// TwinCAT 3 PLC project PLC
// ProgramVersion: 3.1.4024.0
// libraries:
//   EfficientIO Communicator, * (EfficientIO)
//   EfficientIO Energy Basic, * (EfficientIO)
//   Lynus Persistent Data V1, * (Lynus AG)
//   Lynus Standards, * (EfficientIO)
//   Tc2_ModbusSrv, * (Beckhoff Automation GmbH)
//   Tc2_Standard, * (Beckhoff Automation GmbH)
//   Tc2_System, * (Beckhoff Automation GmbH)
//   Tc2_TcpIp, * (Beckhoff Automation GmbH)
//   Tc2_Utilities, * (Beckhoff Automation GmbH)
//   Tc3_Module, * (Beckhoff Automation GmbH)
//   EfficientIO ModbusTCP,1.0.0.9,EfficientIO
// project tree:
//   / FastTask.TcTTO, MiddleTask.TcTTO, SlowTask.TcTTO
//   FB/ fb_Convert4BytesToLreal.TcPOU, FB_IntervalBit.TcPOU (not stored), FB_TCPModbusRequest_PV.TcPOU, FB_TCPModbusRequest_PV_Huawei_inclWrite.TcPOU, FB_TCPModbusRequest_PV_Huawei_inclWrite_oneTurn.TcPOU
//   POUs/ prgBattery.TcPOU, prgComEffIO.TcPOU, prgCS.TcPOU, prgEM.TcPOU, prgEMS.TcPOU, prgGrid.TcPOU, prgPersistent.TcPOU, prgPV_shared.TcPOU, prgPV_separate.TcPOU, prgPV.TcPOU, prgRWEffIO.TcPOU, prgVarEffIO.TcPOU
// real-time tasks:
//   TASK FastTask: cycle T#5ms, priority 19, ADS port 351
//   TASK MiddleTask: cycle T#10ms, priority 20, ADS port 352
//   TASK SlowTask: cycle T#20ms, priority 21, ADS port 353
// I/O:
//   DEVICE Gerät 2 (CX-BK)
//     Box 1 (CX-BK)
// variable links:
//   PLC/PLC Instance <-> Device 2 (CX-BK)/Box 1 (CX-BK)
//     FastTask Inputs/prgGrid.fbKBusState.uiKBusState_OUT <-> Inputs/State
//     MiddleTask Inputs/prgGrid.fbEM1.fbKL3403.byStateCH1 <-> Term 4 (KL3403)/Channel 1/Status
//     MiddleTask Inputs/prgGrid.fbEM1.fbKL3403.byStateCH2 <-> Term 4 (KL3403)/Channel 2/Status
//     MiddleTask Inputs/prgGrid.fbEM1.fbKL3403.byStateCH3 <-> Term 4 (KL3403)/Channel 3/Status
//     MiddleTask Inputs/prgGrid.fbEM1.fbKL3403.iDataInCH1 <-> Term 4 (KL3403)/Channel 1/Daten Ein
//     MiddleTask Inputs/prgGrid.fbEM1.fbKL3403.iDataInCH2 <-> Term 4 (KL3403)/Channel 2/Daten Ein
//     MiddleTask Inputs/prgGrid.fbEM1.fbKL3403.iDataInCH3 <-> Term 4 (KL3403)/Channel 3/Daten Ein
//     MiddleTask Outputs/prgGrid.fbEM1.fbKL3403.byCntrCH1 <-> Term 4 (KL3403)/Channel 1/Kontrolle
//     MiddleTask Outputs/prgGrid.fbEM1.fbKL3403.byCntrCH2 <-> Term 4 (KL3403)/Channel 2/Kontrolle
//     MiddleTask Outputs/prgGrid.fbEM1.fbKL3403.byCntrCH3 <-> Term 4 (KL3403)/Channel 3/Kontrolle

CONFIGURATION PLC
    RESOURCE PLC ON TwinCAT3
        TASK FastTask(INTERVAL := T#5ms, PRIORITY := 19);
        TASK MiddleTask(INTERVAL := T#10ms, PRIORITY := 20);
        TASK SlowTask(INTERVAL := T#20ms, PRIORITY := 21);
        PROGRAM prgPersistent WITH FastTask : prgPersistent;
        PROGRAM prgRWEffIO WITH FastTask : prgRWEffIO;
        PROGRAM prgVarEffIO WITH FastTask : prgVarEffIO;
        PROGRAM prgGrid WITH MiddleTask : prgGrid;
        PROGRAM prgEMS WITH MiddleTask : prgEMS;
        PROGRAM prgCS WITH MiddleTask : prgCS;
        PROGRAM prgEM WITH MiddleTask : prgEM;
        PROGRAM prgBattery WITH MiddleTask : prgBattery;
        PROGRAM prgPV WITH MiddleTask : prgPV;
        PROGRAM prgComEffIO WITH SlowTask : prgComEffIO;
    END_RESOURCE
END_CONFIGURATION

// ---- POUs/prgPersistent.TcPOU
PROGRAM prgPersistent
VAR
	fbUSV		: FB_WritePersistentData_CX81xx;
	
	fb_Reboot		: NT_reboot;
	m_Reboot		: BOOL:=FALSE;
	
	uinit_KbusState: UINT;						//{#lynus.ag#()}
END_VAR

fbUSV(
	eSaveModeData:= eUSVSaveMode.eSaveOnBoth, 
	bLoadPersistentDataOk=> , 
	bPowerFailDetect=> , 
	bError=> , 
	bySaveProcess=> , 
	dwStorageLast24h=> , 
	udiErrorCode=> );
	
	
fb_Reboot(	netid := '',
			delay := 2,
			start := m_Reboot);
	
uinit_KbusState := prgGrid.fbKBusState.uiKBusState_OUT;

END_PROGRAM

// ---- POUs/prgGrid.TcPOU
PROGRAM prgGrid
VAR
	fbKBusState					: FB_K_Bus_State;
	fbEM1						: FB_EM_Beckhoff_KL3403;
	lrPowerGrid					: LREAL;							//{#lynus.ag#()}
	lrPowerEM1_1				: LREAL;							//{#lynus.ag#()}
	lrPowerEM1_2				: LREAL;							//{#lynus.ag#()}
	lrPowerEM1_3				: LREAL;							//{#lynus.ag#()}
	lrCounterGridCon			: LREAL;							//{#lynus.ag#()}
	lrCounterGridProd			: LREAL;							//{#lynus.ag#()}
	lr_GridVoltageL1N_V			: LREAL;							//{#lynus.ag#()}
	lr_GridVoltageL2N_V			: LREAL;							//{#lynus.ag#()}
	lr_GridVoltageL3N_V			: LREAL;							//{#lynus.ag#()}

	lrReactivePowerGrid			: LREAL;							//{#lynus.ag#()}
	lrApparentPowerGrid			: LREAL;							//{#lynus.ag#()}
	fbGrid: FB_Grid_Power;
	lrPowerGrid_cons			: LREAL;							//{#lynus.ag#()}
	lrPowerGrid_prod			: LREAL;							//{#lynus.ag#()}
	lrHouse						: LREAL;							//{#lynus.ag#()}
	
END_VAR

VAR PERSISTENT
	rSizeGridDelivery			: REAL;								//{#lynus.ag#()}
	rSizeGridConn				: REAL;								//{#lynus.ag#()}
END_VAR

//The mapping of this function must be linked with the K-Bus State in the E/A Part
fbKBusState(	uiKBusState_OUT=> , 	
				b_Kbus_notOk=> , 
				word_ErrorCount=> );

//The mapping of this function must be linked with the KL3403 in the E/A Part
//UV1
fbEM1(
	bEnable:= TRUE, 
	bChannel1Invers:= FALSE,				//Invert power data when transformer are mounted upside down
	bChannel2Invers:= FALSE,
	bChannel3Invers:= FALSE,
	uiCurrentTransformerRatioL1:= 1500, // 30 0 / 1 A CTs mounted
	uiCurrentTransformerRatioL2:= 1500, 
	uiCurrentTransformerRatioL3:= 1500, 
	uiKBusState_IN:= fbKBusState.uiKBusState_OUT, 
	stDataEMPower=> , 
	stDataEMCounter=> , 
	stDataEMPowerRealTime=> , 
	stDataEMCounterRealTime=> , 
	diNrOfEM_OUT=> );

lrPowerGrid := fbEM1.stDataEMPower.lrPowerTotal;
lrCounterGridCon := fbEM1.stDataEMCounter.lrTotalCounterEnergy_Consumption;	
lrCounterGridProd := fbEM1.stDataEMCounter.lrTotalCounterEnergy_Production;	
lrPowerEM1_1 := fbEM1.stDataEMPower.lrPowerL1;
lrPowerEM1_2 := fbEM1.stDataEMPower.lrPowerL2;
lrPowerEM1_3 := fbEM1.stDataEMPower.lrPowerL3;

lrReactivePowerGrid:=fbEM1.stDataEMPower.lrReactivePowerTotal;
lrApparentPowerGrid:=fbEM1.stDataEMPower.lrApparentPowerTotal;

lr_GridVoltageL1N_V:=fbEM1.stDataEMPower.lrVoltageL1N;
lr_GridVoltageL2N_V:=fbEM1.stDataEMPower.lrVoltageL2N;
lr_GridVoltageL3N_V:=fbEM1.stDataEMPower.lrVoltageL3N;

fbGrid(
	bEnable:= TRUE, 
	diNrOfEMS_IN:= prgEMS.fbEMS.diNrOfEMS_OUT, 
	diNrOfEM_IN_Grid:= 	fbEM1.diNrOfEM_OUT,			//prgBattery.fbBattery.diNrOfEM_OUT_Grid, 
	rSizeGridConn:= rSizeGridConn, 
	stDataGrid=> , 
	diNrOfGrid_OUT=> );

lrPowerGrid_cons 	:= 	fbEM1.stDataEMPower.lrPowerConsumption;
lrPowerGrid_prod	:= 	fbEM1.stDataEMPower.lrPowerProduction;

lrHouse := lrPowerGrid + prgPV.lrPowerPV - prgCS.lrPowerCS + prgBattery.lrPowerBattery + prgEM.lrPower_Fuse - prgEM.lrPower_Fuse_EM2 - prgEM.lrPower_Fuse_EM3;

END_PROGRAM

// ---- POUs/prgEMS.TcPOU
PROGRAM prgEMS
VAR PERSISTENT
	byMaxDepthOfDischrgEPO		: BYTE;							//{#lynus.ag#()}
	byPrioMinChrgBattSOCInEPO	: BYTE;							//{#lynus.ag#()}
	byResChrgfromGridToBatt		: BYTE;							//{#lynus.ag#()}
	byReserveSOCEPO				: BYTE;							//{#lynus.ag#()}
	uiUpdateTime				: UINT;							//{#lynus.ag#()}
	bEnableEMS					: BOOL;							//{#lynus.ag#()}
	bAllowChrgFromGrid			: BOOL;							//{#lynus.ag#()}
	bActivateMainFuse			: BOOL;							//{#lynus.ag#()}
	rMainFuseCSEMS				: REAL;							//{#lynus.ag#()}
	iOperationModeEMS			: INT;							//{#lynus.ag#()}
	by_MinSOC_AdaptiveLC		: BYTE;							//{#lynus.ag#()}
END_VAR
VAR
	fbEMS						: FB_EMS_V12;
	bIsEnableEMS				: BOOL;							//{#lynus.ag#()}
	bStateAllowChrgFromGrid		: BOOL;							//{#lynus.ag#()}
	bHPActivate					: BOOL;							//{#lynus.ag#()}
	bControllingState			: BOOL;							//{#lynus.ag#()}
	bSActivateMainFuse			: BOOL;							//{#lynus.ag#()}
	iMessageEMS					: INT;							//{#lynus.ag#()}
	rHeartbeatEMS				: REAL;							//{#lynus.ag#()}
	rErrorWarningEMS			: REAL;							//{#lynus.ag#()}
	rReadyEMS					: REAL;							//{#lynus.ag#()}
	rNewBatteryPowerEMS			: REAL;							//{#lynus.ag#()}
	b_Chargefor3Hours			: BOOL;							//{#lynus.ag#()}
	b_Chargefor3Hours_Active	: BOOL;							//{#lynus.ag#()}
	b_Chargefor1Hour			: BOOL;							//{#lynus.ag#()}
	b_Chargefor1Hour_Active		: BOOL;							//{#lynus.ag#()}
	ton_ChargeTimer_3hours		: ton;
	ton_ChargeTimer_1hour		: ton;
	rs_charge_3hours			: rs;
	rs_charge_1hour				: rs;
	r_trig_Charge_3hours		: R_trig;
	r_trig_Charge_1hour			: R_trig;
	fb_Meter	:	FB_EM_Electric_3P_Ext_Input;
	iOperationModeEMS_actual			: INT;							//{#lynus.ag#()}
	di_temp : DINT;
	m_ZeroPowerRegulationActive: BOOL:=FALSE;						//{#lynus.ag#()}
	timer_CarConnected_CSPowerlow: Ton;

END_VAR

fbEMS.stSetupEMS.bAllowChrgFromGrid := bAllowChrgFromGrid;
fbEMS.stSetupEMS.byMaxDepthOfDischrgEPO := byMaxDepthOfDischrgEPO;
fbEMS.stSetupEMS.byResChrgfromGridToBatt := byResChrgfromGridToBatt;
fbEMS.stSetupEMS.byPrioMinChrgBattSOCInEPO := byPrioMinChrgBattSOCInEPO;
fbEMS.stSetupEMS.byReserveSOCEPO := SEL(b_Chargefor3Hours_Active OR b_Chargefor1Hour_Active,byReserveSOCEPO,100);
fbEMS.stSetupEMS.rSizeMainFuseCS := rMainFuseCSEMS;
fbEMS.stSetupEMS.uiUpdateTime := uiUpdateTime;
fbEMS.stSetupEMS.bEnableMainFuseFunction := bActivateMainFuse;

IF iOperationModeEMS = 0 THEN 
	fbEMS.eOperationMode_Ext := E_OperatingMode_EMS.eAllOff;
ELSIF iOperationModeEMS = 1 THEN 
	fbEMS.eOperationMode_Ext := E_OperatingMode_EMS.eSelfConsumption;	
ELSIF iOperationModeEMS = 2 THEN 
	fbEMS.eOperationMode_Ext := E_OperatingMode_EMS.ePeakLoadCapping;
ELSIF iOperationModeEMS = 3 THEN 
	fbEMS.eOperationMode_Ext := E_OperatingMode_EMS.eLoadManagement;			
ELSIF iOperationModeEMS = 4 THEN 
	fbEMS.eOperationMode_Ext := E_OperatingMode_EMS.eAdaptiveLoadControl;		
END_IF
di_temp := fbEMS.diNumberOfActiveBatterys;

fbEMS(
	diNrOfEM_IN_ECS:= , 
	stSetupEMS:= , 
	eOperationMode_Ext:= , 
	eSpeedModeBackendController:= E_SpeedModeBackendController_EMS.eSlow,	//.efast, 
	eSpeedModeLocalController:= E_SpeedModeLocalController_EMS.eSlow,    //efast,
	bZeroPowerRegulation	:= m_ZeroPowerRegulationActive, 
	by_MinSOC_AdaptiveLC:= by_MinSOC_AdaptiveLC, 
	bActivateHP:= bHPActivate, 
	bControllingState:= TRUE, //bControllingState, 
	rHeartbeat:= rHeartbeatEMS, 
	rErrorWarning:= rErrorWarningEMS, 
	rEnergyOptReady:= rReadyEMS, 
	rNewBattPower:= rNewBatteryPowerEMS,
	b_AnyCarConnected:= prgCS.bCarConnected and not timer_CarConnected_CSPowerlow.Q ,  
	eMessageEMS=> iMessageEMS, 
	bStateEnable=> bIsEnableEMS, 
	bStateAllowChrgFromGrid=> bStateAllowChrgFromGrid, 
	bMissingPowerData=> , 
	bSurplusAvailable=> , 
	byProgress=> , 
	uiState_OUT=> , 
	diNrOfEMS_OUT=> , 
	arrMinPrioReached=> , 
	arrMaxPrioReached=> );
	
bSActivateMainFuse := fbEMS.stSetupEMS.bEnableMainFuseFunction;	
iOperationModeEMS_actual := fbEMS.eOperationMode;

// charge for 3 hours
r_trig_Charge_3hours (clk := b_Chargefor3Hours);
r_trig_Charge_1hour (clk := b_Chargefor1Hour);


rs_charge_3hours	(	Set := r_trig_Charge_3hours.Q ,
						Reset1 := ton_ChargeTimer_3hours.Q OR (rs_Charge_3hours.Q1 AND r_trig_Charge_3hours.Q),
						Q1 => b_Chargefor3Hours_Active);
rs_charge_1hour		(	Set := r_trig_Charge_1hour.Q ,
						Reset1 := ton_ChargeTimer_1hour.Q OR (rs_Charge_1hour.Q1 AND r_trig_Charge_1hour.Q),
						Q1 => b_Chargefor1Hour_Active);			
ton_ChargeTimer_3hours	( 	IN := rs_charge_3hours.Q1,
							PT := T#3H,
							Q => );
ton_ChargeTimer_1hour	( 	IN := rs_charge_1hour.Q1,
							PT := T#1H,
							Q => );
	

timer_CarConnected_CSPowerlow( 	IN := prgCS.bCarConnected AND prgCS.lrPowerCS < 2,	// required to get out of zero power regulation if a car is connected all night long
								PT := T#10M);
							
m_ZeroPowerRegulationActive := prgCS.bCarConnected AND NOT timer_CarConnected_CSPowerlow.Q;
	

fb_Meter(
	bEnable:= TRUE, 
	bPowerDataInvers:= , 
	bErrorExt:= , 
	bWarningExt:= , 
	lrTotalCounterEnergy_Consumption:= , 
	lrTotalCounterEnergy_Production:= , 
	lrCounterEnergyT1_Consumption:= , 
	lrCounterEnergyT2_Consumption:= , 
	lrCounterEnergyT1_Production:= , 
	lrCounterEnergyT2_Production:= , 
	lrCurrentL1:= , 
	lrVoltageL1N:= , 
	lrVoltageL1L2:= , 
	lrPowerL1:= , 
	lrCurrentL2:= , 
	lrVoltageL2N:= , 
	lrVoltageL2L3:= , 
	lrPowerL2:= , 
	lrCurrentL3:= , 
	lrVoltageL3N:= , 
	lrVoltageL3L1:= , 
	lrPowerL3:= , 
	lrPowerTotal:= prgEM.lrPower_Fuse,
	lrFrequency:= , 
	lrReactivePowerTotal:= , 
	lrApparentPowerTotal:= , 
	stDataEMPower=> , 
	stDataEMCounter=> , 
	diNrOfEM_OUT=> );		// da gehört was hin, damit er auf die fuseline regeln kann

END_PROGRAM

// ---- POUs/prgCS.TcPOU
PROGRAM prgCS
VAR PERSISTENT
	bEnabledCS				: BOOL;									//{#lynus.ag#()}
	byPrioCS				: BYTE;									//{#lynus.ag#()}
	bySOC_E_CS				: BYTE;									//{#lynus.ag#()}
	bySOC_D_CS				: BYTE;									//{#lynus.ag#()}
	byMinPowerCS			: BYTE;									//{#lynus.ag#()}
	rMaxPowerCS				: REAL;									//{#lynus.ag#()}
	lrCounterCS				: LREAL;								//{#lynus.ag#()}
	bManualyOn				: BOOL;									//{#lynus.ag#()}
	byMinPower				: BYTE;									//{#lynus.ag#()}
	byManualyTargetPower	: BYTE;									//{#lynus.ag#()}
	m_ChargingLimit			: BOOL;									//{#lynus.ag#()}
	bOnEmergPowerOff		: BOOL;									//{#lynus.ag#()}
END_VAR
VAR
	fbCS					: FB_ECS_Alpitronic_Hypercharger;
	fbCSCounter				: FB_EnergyCounter;
	bIsEnabledCS			: BOOL;									//{#lynus.ag#()}
	byErrorWarningCS		: BYTE;									//{#lynus.ag#()}
	byStateMinPowerCS		: BYTE;									//{#lynus.ag#()}
	rTargetPowerCS			: REAL;									//{#lynus.ag#()}
	bCarConnected			: BOOL;									//{#lynus.ag#()}
	rChrgTime				: REAL;									//{#lynus.ag#()}
	lrPowerCS				: LREAL;								//{#lynus.ag#()}
	bSManualyOn				: BOOL;									//{#lynus.ag#()}
	bySManualyTargetPower	: BYTE;									//{#lynus.ag#()}
	str_IP: STRING(15):='172.16.127.151';
	rSOC_1					: REAL;									//{#lynus.ag#()}
	rSOC_2					: REAL;									//{#lynus.ag#()}
	bSOnEmergPowerOff		: BOOL;									//{#lynus.ag#()}
END_VAR

fbCS.stSetupECS.byDisableSOC := bySOC_D_CS;
fbCS.stSetupECS.byEnableSOC := bySOC_E_CS;
fbCS.stSetupECS.byPriority := byPrioCS;
fbCS.stSetupECS.rMaxPower := rMaxPowerCS;
fbCS.stSetupECS.byCSMinPower := byMinPowerCS;
fbCS.stSetupECS.bManualyOn := bManualyOn;
fbCS.stSetupECS.byManualyTargetPower := byManualyTargetPower;
fbCS.stSetupECS.byCSMinPower := byMinPower;
fbCS.stSetupECS.bOnEmergPowerOff := bOnEmergPowerOff;

fbCS(
	bEnable:= bEnabledCS, 
	bPowerDataInvers:= ,  
	byUnitID:= 1,				//Allways 1 
	diNrOfEMS_IN:= prgEMS.fbEMS.diNrOfEMS_OUT, 
	diNrOfEM_IN_CS:= , 
	sIPAdress:= str_IP, 
	stSetupECS:= , 
	stDataECS=> , 
	diNrOfECS_OUT=> );

bIsEnabledCS := fbCS.stDataECS.bEnabled;
byStateMinPowerCS := fbCS.stDataECS.bySCSMinPower;
rTargetPowerCS := fbCS.stDataECS.rTargetPower;	
byErrorWarningCS := fbCS.stDataECS.byErrorWarning;
bCarConnected := fbCS.stDataECS.bCarConnected;
rChrgTime := MAX(fbCS.stDataECS.arrChargingTimeInMin[1],fbCS.stDataECS.arrChargingTimeInMin[2]);
lrPowerCS := fbCS.stDataECS.lrTotalPower;
bSManualyOn := fbCS.stDataECS.bSManualyOn;
bSOnEmergPowerOff := fbCS.stDataECS.bSOnEmergPowerOff;

bySManualyTargetPower := fbCS.stDataECS.bySManualyTargetPower;
rSOC_1	:= DWORD_TO_REAL(fbCS.stDataECS.arrSocketSOCCar[1]);
rSOC_2	:= DWORD_TO_REAL(fbCS.stDataECS.arrSocketSOCCar[2]);						

// EnergyCounter
fbCSCounter(
	byActiveTariff:= 1, 
	lrPowerInput:= lrPowerCS, 
	lrTotalCounterEnergy_Consumption=> );
	
IF fbCSCounter.lrTotalCounterEnergy_Consumption > lrCounterCS THEN  	
	lrCounterCS := fbCSCounter.lrTotalCounterEnergy_Consumption;
END_IF

END_PROGRAM

// ---- POUs/prgEM.TcPOU
PROGRAM prgEM
VAR
	// Meter1 - Halle Verteiler
	fb_External_Meter			: fb_EM24_DIN;
	str_IP: STRING(15)			:= '172.16.127.51'	;
	
	lrPower_Fuse				: LREAL;							//{#lynus.ag#()}
	lrPower_Fuse_1				: LREAL;							//{#lynus.ag#()}
	lrPower_Fuse_2				: LREAL;							//{#lynus.ag#()}
	lrPower_Fuse_3				: LREAL;							//{#lynus.ag#()}
	lrCurrent_Fuse_1			: LREAL;							//{#lynus.ag#()}
	lrCurrent_Fuse_2			: LREAL;							//{#lynus.ag#()}
	lrCurrent_Fuse_3			: LREAL;							//{#lynus.ag#()}
	lrCounter_Fuse_Con			: LREAL;							//{#lynus.ag#()}
	lrCounter_Fuse_Prod			: LREAL;							//{#lynus.ag#()}
	lr_Voltage_Fuse_L1N_V		: LREAL;							//{#lynus.ag#()}
	lr_Voltage_Fuse_L2N_V		: LREAL;							//{#lynus.ag#()}
	lr_Voltage_Fuse_L3N_V		: LREAL;							//{#lynus.ag#()}
	lr_Voltage_Fuse_L1L2_V		: LREAL;							//{#lynus.ag#()}
	lr_Voltage_Fuse_L2L3_V		: LREAL;							//{#lynus.ag#()}
	lr_Voltage_Fuse_L3L1_V		: LREAL;							//{#lynus.ag#()}

	lrReactivePowerFuse			: LREAL;							//{#lynus.ag#()}
	lrApparentPowerFuse			: LREAL;							//{#lynus.ag#()}
	m_invert					: BOOL:=TRUE;
	
	
	// Meter2 - 3. Stock
	fb_External_Meter_2				: fb_EM24_DIN;
	str_IP_EM2						: STRING(15):= '172.16.127.52'	;
	
	lrPower_Fuse_EM2				: LREAL;							//{#lynus.ag#()}
	lrPower_Fuse_1_EM2				: LREAL;							//{#lynus.ag#()}
	lrPower_Fuse_2_EM2				: LREAL;							//{#lynus.ag#()}
	lrPower_Fuse_3_EM2				: LREAL;							//{#lynus.ag#()}
	lrCurrent_Fuse_1_EM2			: LREAL;							//{#lynus.ag#()}
	lrCurrent_Fuse_2_EM2			: LREAL;							//{#lynus.ag#()}
	lrCurrent_Fuse_3_EM2			: LREAL;							//{#lynus.ag#()}
	lrCounter_Fuse_Con_EM2			: LREAL;							//{#lynus.ag#()}
	lrCounter_Fuse_Prod_EM2			: LREAL;							//{#lynus.ag#()}
	lr_Voltage_Fuse_L1N_V_EM2		: LREAL;							//{#lynus.ag#()}
	lr_Voltage_Fuse_L2N_V_EM2		: LREAL;							//{#lynus.ag#()}
	lr_Voltage_Fuse_L3N_V_EM2		: LREAL;							//{#lynus.ag#()}
	lr_Voltage_Fuse_L1L2_V_EM2		: LREAL;							//{#lynus.ag#()}
	lr_Voltage_Fuse_L2L3_V_EM2		: LREAL;							//{#lynus.ag#()}
	lr_Voltage_Fuse_L3L1_V_EM2		: LREAL;							//{#lynus.ag#()}

	lrReactivePowerFuse_EM2			: LREAL;							//{#lynus.ag#()}
	lrApparentPowerFuse_EM2			: LREAL;							//{#lynus.ag#()}
	m_invert_EM2					: BOOL:=FALSE;
	
	
	// Meter3 - EG
	fb_External_Meter_3				: fb_EM24_DIN;
	str_IP_EM3						: STRING(15):= '172.16.127.53'	;
	
	lrPower_Fuse_EM3				: LREAL;							//{#lynus.ag#()}
	lrPower_Fuse_1_EM3				: LREAL;							//{#lynus.ag#()}
	lrPower_Fuse_2_EM3				: LREAL;							//{#lynus.ag#()}
	lrPower_Fuse_3_EM3				: LREAL;							//{#lynus.ag#()}
	lrCurrent_Fuse_1_EM3			: LREAL;							//{#lynus.ag#()}
	lrCurrent_Fuse_2_EM3			: LREAL;							//{#lynus.ag#()}
	lrCurrent_Fuse_3_EM3			: LREAL;							//{#lynus.ag#()}
	lrCounter_Fuse_Con_EM3			: LREAL;							//{#lynus.ag#()}
	lrCounter_Fuse_Prod_EM3			: LREAL;							//{#lynus.ag#()}
	lr_Voltage_Fuse_L1N_V_EM3		: LREAL;							//{#lynus.ag#()}
	lr_Voltage_Fuse_L2N_V_EM3		: LREAL;							//{#lynus.ag#()}
	lr_Voltage_Fuse_L3N_V_EM3		: LREAL;							//{#lynus.ag#()}
	lr_Voltage_Fuse_L1L2_V_EM3		: LREAL;							//{#lynus.ag#()}
	lr_Voltage_Fuse_L2L3_V_EM3		: LREAL;							//{#lynus.ag#()}
	lr_Voltage_Fuse_L3L1_V_EM3		: LREAL;							//{#lynus.ag#()}

	lrReactivePowerFuse_EM3			: LREAL;							//{#lynus.ag#()}
	lrApparentPowerFuse_EM3			: LREAL;							//{#lynus.ag#()}
	m_invert_EM3					: BOOL:=FALSE;
	
END_VAR

// Meter1 - Halle Verteiler
fb_External_Meter(
	m_Enable:= TRUE, 
	str_IPAdress:= str_IP, 
	real_RealPower_kW=> lrPower_Fuse, 
	real_RealPowerL1_kW=> lrPower_Fuse_1, 
	real_RealPowerL2_kW=> lrPower_Fuse_2, 
	real_RealPowerL3_kW=> lrPower_Fuse_3, 
	real_ReactivePower_kVAr=> lrReactivePowerFuse, 
	real_ApparentPower_kVA=> lrApparentPowerFuse, 
	real_Frequency_Hz=> , 
	real_VoltageL1N_V=> lr_Voltage_Fuse_L1N_V, 
	real_VoltageL2N_V=> lr_Voltage_Fuse_L2N_V, 
	real_VoltageL3N_V=> lr_Voltage_Fuse_L3N_V, 
	real_VoltageL1L2_V=> lr_Voltage_Fuse_L1L2_V, 
	real_VoltageL2L3_V=> lr_Voltage_Fuse_L2L3_V, 
	real_VoltageL3L1_V=> lr_Voltage_Fuse_L3L1_V, 
	real_CurrentL1_A=> lrCurrent_Fuse_1, 
	real_CurrentL2_A=> lrCurrent_Fuse_2, 
	real_CurrentL3_A=> lrCurrent_Fuse_3, 
	real_EnergyTotal_Import_kWh=> , 
	real_EnergyTotal_Export_kWh=> , 
	real_EnergyTotal_ExportT1_kWh=> , 
	real_EnergyTotal_ExportT2_kWh=> , 
	real_EnergyTotal_ExportT3_kWh=> , 
	real_EnergyTotal_ExportT4_kWh=> , 
	m_PollSuccessful=> , 
	udint_Error_ID=> );
IF m_invert THEN
	lrPower_Fuse_1 		:= -lrPower_Fuse_1 		;
    lrPower_Fuse_2      := -lrPower_Fuse_2      ;
    lrPower_Fuse_3      := -lrPower_Fuse_3      ;
	lrPower_Fuse        := -lrPower_Fuse        ;
	lrCurrent_Fuse_1    := -lrCurrent_Fuse_1    ;
    lrCurrent_Fuse_2    := -lrCurrent_Fuse_2    ;
    lrCurrent_Fuse_3    := -lrCurrent_Fuse_3    ;
END_IF	
IF lrPower_Fuse > 0 THEN 
	lrCounter_Fuse_Con := lrPower_Fuse;
	lrCounter_Fuse_Prod := 0;
ELSE
	lrCounter_Fuse_Prod := lrPower_Fuse;
	lrCounter_Fuse_Con := 0;
END_IF


// Meter2 - 3. Stock
fb_External_Meter_2(
	m_Enable:= TRUE, 
	str_IPAdress:= str_IP_EM2, 
	real_RealPower_kW=> lrPower_Fuse_EM2, 
	real_RealPowerL1_kW=> lrPower_Fuse_1_EM2, 
	real_RealPowerL2_kW=> lrPower_Fuse_2_EM2, 
	real_RealPowerL3_kW=> lrPower_Fuse_3_EM2, 
	real_ReactivePower_kVAr=> lrReactivePowerFuse_EM2, 
	real_ApparentPower_kVA=> lrApparentPowerFuse_EM2, 
	real_Frequency_Hz=> , 
	real_VoltageL1N_V=> lr_Voltage_Fuse_L1N_V_EM2, 
	real_VoltageL2N_V=> lr_Voltage_Fuse_L2N_V_EM2, 
	real_VoltageL3N_V=> lr_Voltage_Fuse_L3N_V_EM2, 
	real_VoltageL1L2_V=> lr_Voltage_Fuse_L1L2_V_EM2, 
	real_VoltageL2L3_V=> lr_Voltage_Fuse_L2L3_V_EM2, 
	real_VoltageL3L1_V=> lr_Voltage_Fuse_L3L1_V_EM2, 
	real_CurrentL1_A=> lrCurrent_Fuse_1_EM2, 
	real_CurrentL2_A=> lrCurrent_Fuse_2_EM2, 
	real_CurrentL3_A=> lrCurrent_Fuse_3_EM2, 
	real_EnergyTotal_Import_kWh=> , 
	real_EnergyTotal_Export_kWh=> , 
	real_EnergyTotal_ExportT1_kWh=> , 
	real_EnergyTotal_ExportT2_kWh=> , 
	real_EnergyTotal_ExportT3_kWh=> , 
	real_EnergyTotal_ExportT4_kWh=> , 
	m_PollSuccessful=> , 
	udint_Error_ID=> );
IF m_invert_EM2 THEN
	lrPower_Fuse_1_EM2 		:= -lrPower_Fuse_1_EM2 		;
    lrPower_Fuse_2_EM2      := -lrPower_Fuse_2_EM2      ;
    lrPower_Fuse_3_EM2      := -lrPower_Fuse_3_EM2      ;
	lrPower_Fuse_EM2        := -lrPower_Fuse_EM2        ;
	lrCurrent_Fuse_1_EM2    := -lrCurrent_Fuse_1_EM2    ;
    lrCurrent_Fuse_2_EM2    := -lrCurrent_Fuse_2_EM2    ;
    lrCurrent_Fuse_3_EM2    := -lrCurrent_Fuse_3_EM2    ;
END_IF	
IF lrPower_Fuse_EM2 > 0 THEN 
	lrCounter_Fuse_Con_EM2 := lrPower_Fuse_EM2;
	lrCounter_Fuse_Prod_EM2 := 0;
ELSE
	lrCounter_Fuse_Prod_EM2 := lrPower_Fuse_EM2;
	lrCounter_Fuse_Con_EM2 := 0;
END_IF


// Meter3 - EG
fb_External_Meter_3(
	m_Enable:= TRUE, 
	str_IPAdress:= str_IP_EM3, 
	real_RealPower_kW=> lrPower_Fuse_EM3, 
	real_RealPowerL1_kW=> lrPower_Fuse_1_EM3, 
	real_RealPowerL2_kW=> lrPower_Fuse_2_EM3, 
	real_RealPowerL3_kW=> lrPower_Fuse_3_EM3, 
	real_ReactivePower_kVAr=> lrReactivePowerFuse_EM3, 
	real_ApparentPower_kVA=> lrApparentPowerFuse_EM3, 
	real_Frequency_Hz=> , 
	real_VoltageL1N_V=> lr_Voltage_Fuse_L1N_V_EM3, 
	real_VoltageL2N_V=> lr_Voltage_Fuse_L2N_V_EM3, 
	real_VoltageL3N_V=> lr_Voltage_Fuse_L3N_V_EM3, 
	real_VoltageL1L2_V=> lr_Voltage_Fuse_L1L2_V_EM3, 
	real_VoltageL2L3_V=> lr_Voltage_Fuse_L2L3_V_EM3, 
	real_VoltageL3L1_V=> lr_Voltage_Fuse_L3L1_V_EM3, 
	real_CurrentL1_A=> lrCurrent_Fuse_1_EM3, 
	real_CurrentL2_A=> lrCurrent_Fuse_2_EM3, 
	real_CurrentL3_A=> lrCurrent_Fuse_3_EM3, 
	real_EnergyTotal_Import_kWh=> , 
	real_EnergyTotal_Export_kWh=> , 
	real_EnergyTotal_ExportT1_kWh=> , 
	real_EnergyTotal_ExportT2_kWh=> , 
	real_EnergyTotal_ExportT3_kWh=> , 
	real_EnergyTotal_ExportT4_kWh=> , 
	m_PollSuccessful=> , 
	udint_Error_ID=> );
IF m_invert_EM3 THEN
	lrPower_Fuse_1_EM3 		:= -lrPower_Fuse_1_EM3 		;
    lrPower_Fuse_2_EM3      := -lrPower_Fuse_2_EM3      ;
    lrPower_Fuse_3_EM3      := -lrPower_Fuse_3_EM3      ;
	lrPower_Fuse_EM3        := -lrPower_Fuse_EM3        ;
	lrCurrent_Fuse_1_EM3    := -lrCurrent_Fuse_1_EM3    ;
    lrCurrent_Fuse_2_EM3    := -lrCurrent_Fuse_2_EM3    ;
    lrCurrent_Fuse_3_EM3    := -lrCurrent_Fuse_3_EM3    ;
END_IF	
IF lrPower_Fuse_EM3 > 0 THEN 
	lrCounter_Fuse_Con_EM3 := lrPower_Fuse_EM3;
	lrCounter_Fuse_Prod_EM3 := 0;
ELSE
	lrCounter_Fuse_Prod_EM3 := lrPower_Fuse_EM3;
	lrCounter_Fuse_Con_EM3 := 0;
END_IF

END_PROGRAM

// ---- POUs/prgPV.TcPOU
PROGRAM prgPV
VAR
	lrPowerPV				: LREAL;				//{#lynus.ag#()}
		// extend or reduce amount of PV Inverters
	lrPowerPV_1				: LREAL;				//{#lynus.ag#()}
	lrPowerPV_2				: LREAL;				//{#lynus.ag#()}
	uint_setPoint_onetenth: UINT;						//{#lynus.ag#()}

	m_shared: BOOL;
END_VAR
VAR PERSISTENT
	lrCounterPV_1				: LREAL;				//{#lynus.ag#()}
	lrCounterPV_2				: LREAL;				//{#lynus.ag#()}
END_VAR

IF m_shared THEN
	prgPV_shared();
	lrPowerPV 				:= prgPV_shared.lrPowerPV;
	lrPowerPV_1 			:= prgPV_shared.lrPowerPV_1;
	lrPowerPV_2 			:= prgPV_shared.lrPowerPV_2;
	uint_setPoint_onetenth 	:= prgPV_shared.uint_setPoint_onetenth;
	lrCounterPV_1			:= prgPV_shared.lrCounterPV_1;
	lrCounterPV_2			:= prgPV_shared.lrCounterPV_2;
ELSE
	prgPV_separate();
	lrPowerPV 				:= prgPV_separate.lrPowerPV;
	lrPowerPV_1 			:= prgPV_separate.lrPowerPV_1;
	lrPowerPV_2 			:= prgPV_separate.lrPowerPV_2;
	uint_setPoint_onetenth 	:= prgPV_separate.uint_setPoint_onetenth;
	lrCounterPV_1			:= prgPV_separate.lrCounterPV_1;
	lrCounterPV_2			:= prgPV_separate.lrCounterPV_2;
END_IF

END_PROGRAM

// ---- POUs/prgPV_shared.TcPOU
PROGRAM prgPV_shared
VAR
	fbPVCounter_1			: FB_EnergyCounter;
	fbPVCounter_2			: FB_EnergyCounter;
	lrPowerPV				: LREAL;				
		// extend or reduce amount of PV Inverters
	lrPowerPV_1				: LREAL;				
	lrPowerPV_2				: LREAL;				

	str_IP: STRING(15) := '172.16.127.240';
	FB_PV_1:FB_TCPModbusRequest_PV_Huawei_inclWrite;	
	FB_PV_2:FB_TCPModbusRequest_PV_Huawei_inclWrite;	
	fb_Meter_1		: FB_EM_Electric_3P_Ext_Input;
	fbPVInt_1		: FB_PV_Power;
	fb_Meter_2		: FB_EM_Electric_3P_Ext_Input;
	fbPVInt_2		: FB_PV_Power;
	

	FB_PID_Inverter :FB_PID;

	uint_setPoint_onetenth: UINT;					

	rPValue: REAL := 0.5;
	udint_IValue: UDINT:=250;
	udint_DValue: UDINT:=30;

	unit_Temp: UINT;
	real_max: REAL:=1000;
	real_min: REAL:=10;

END_VAR
VAR PERSISTENT
	lrCounterPV_1				: LREAL;				
	lrCounterPV_2				: LREAL;				
	m_Direction: BOOL := true;
END_VAR

FB_PV_1(
	b_Enable:= , 
	by_slave_ID:= 1, 
	str_IPAdress:= str_ip, 
	uint_SetPoint_onetenth:= uint_setPoint_onetenth, 
	lreal_RealPower_kW=> lrPowerPV_1,  );


fbPVCounter_1(	byActiveTariff := 1,	
	
				lrPowerInput := 0-lrPowerPV_1,
				lrTotalCounterEnergy_Production => lrCounterPV_1);


FB_PV_2(
	b_Enable:= , 
	by_slave_ID:= 2, 
	str_IPAdress:= str_ip, 
	uint_SetPoint_onetenth:= uint_setPoint_onetenth, 
	lreal_RealPower_kW=> lrPowerPV_2,  );


fbPVCounter_2(	byActiveTariff := 1,	
				lrPowerInput := 0-lrPowerPV_2,
				lrTotalCounterEnergy_Production => lrCounterPV_2);

lrPowerPV := lrPowerPV_1 + lrPowerPV_2;

fbPVInt_1(
	bEnable:= TRUE, 
	bPowerDataInvers:= , 
	diNrOfEM_IN_PV:= fb_Meter_1.diNrOfEM_OUT, 
	stDataPv=> , 
	diNrOfPv_OUT=> );
	
fb_Meter_1(
	bEnable:= TRUE, 
	bPowerDataInvers:= , 
	bErrorExt:= , 
	bWarningExt:= , 
	lrTotalCounterEnergy_Consumption:= , 
	lrTotalCounterEnergy_Production:= , 
	lrCounterEnergyT1_Consumption:= , 
	lrCounterEnergyT2_Consumption:= , 
	lrCounterEnergyT1_Production:= , 
	lrCounterEnergyT2_Production:= , 
	lrCurrentL1:= , 
	lrVoltageL1N:= , 
	lrVoltageL1L2:= , 
	lrPowerL1:= , 
	lrCurrentL2:= , 
	lrVoltageL2N:= , 
	lrVoltageL2L3:= , 
	lrPowerL2:= , 
	lrCurrentL3:= , 
	lrVoltageL3N:= , 
	lrVoltageL3L1:= , 
	lrPowerL3:= , 
	lrPowerTotal:= lrPowerPV_1,
	lrFrequency:= , 
	lrReactivePowerTotal:= , 
	lrApparentPowerTotal:= , 
	stDataEMPower=> , 
	stDataEMCounter=> , 
	diNrOfEM_OUT=> );

	

fbPVInt_2(
	bEnable:= TRUE, 
	bPowerDataInvers:= , 
	diNrOfEM_IN_PV:= fb_Meter_2.diNrOfEM_OUT, 
	stDataPv=> , 
	diNrOfPv_OUT=> );
	
fb_Meter_2(	
	bEnable:= TRUE, 
	bPowerDataInvers:= , 
	bErrorExt:= , 
	bWarningExt:= , 
	lrTotalCounterEnergy_Consumption:= , 
	lrTotalCounterEnergy_Production:= , 
	lrCounterEnergyT1_Consumption:= , 
	lrCounterEnergyT2_Consumption:= , 
	lrCounterEnergyT1_Production:= , 
	lrCounterEnergyT2_Production:= , 
	lrCurrentL1:= , 
	lrVoltageL1N:= , 
	lrVoltageL1L2:= , 
	lrPowerL1:= , 
	lrCurrentL2:= , 
	lrVoltageL2N:= , 
	lrVoltageL2L3:= , 
	lrPowerL2:= , 
	lrCurrentL3:= , 
	lrVoltageL3N:= , 
	lrVoltageL3L1:= , 
	lrPowerL3:= , 
	lrPowerTotal:= lrPowerPV_2,
	lrFrequency:= , 
	lrReactivePowerTotal:= , 
	lrApparentPowerTotal:= , 
	stDataEMPower=> , 
	stDataEMCounter=> , 
	diNrOfEM_OUT=> );

	
FB_PID_Inverter(
		bEnable:= TRUE, 
		rSetpoint:= -prgGrid.rSizeGridDelivery, 
		udiIValue:= udint_IValue, 
		udiDValue:= udint_DValue, 
		udiDamping:= 0, 
		rPValue:= rPValue, 
		rMaxValue:= real_max, 
		rMinValue:= real_min, 
		rNeutralZone:= 1, 
		bDirection:= m_Direction, 
		rActualValue:=  LREAL_TO_REAL(prgGrid.fbEM1.stDataEMPowerRealTime.lrPowerTotal),
		rQController=> );
uint_setPoint_onetenth := REAL_TO_UINT(FB_PID_Inverter.rQController);

END_PROGRAM

// ---- FB/FB_TCPModbusRequest_PV_Huawei_inclWrite.TcPOU
FUNCTION_BLOCK FB_TCPModbusRequest_PV_Huawei_inclWrite
VAR_INPUT
	b_Enable: BOOL;
	by_slave_ID	:BYTE;
	str_IPAdress: STRING(15);
	uint_SetPoint_onetenth	:UINT;
END_VAR
VAR_OUTPUT

	lreal_RealPower_kW:LREAL;
	lreal_Voltage_L1L2_V: LREAL;
	lreal_Voltage_L2L3_V: LREAL;
	lreal_Voltage_L3L1_V: LREAL;
	lreal_Voltage_L1_V: LREAL;
	lreal_Voltage_L2_V: LREAL;
	lreal_Voltage_L3_V: LREAL;
	lreal_Current_L1_A: LREAL;
	lreal_Current_L2_A: LREAL;
	lreal_Current_L3_A: LREAL;
	lreal_PeakPowerDay_kW: LREAL;
	lreal_Power2_kW: LREAL;
	lreal_ReactivePower_kVAr: LREAL;
	lreal_PowerFactor: LREAL;
	lreal_Frequency_Hz: LREAL;
	lreal_Efficiency: LREAL;
	lreal_InternalTemperature_C: LREAL;
	lreal_IsolationResistance_MOhm: LREAL;
END_VAR
VAR
	i_State:INT;
	FB_SocketConnect : FB_SocketConnect;
	hSocket : T_HSOCKET;
	FB_SocketSend : FB_SocketSend;
	FB_SocketReceive : FB_SocketReceive;
	byteSendString : ARRAY[1..12] OF BYTE;
	FB_CloseSockets: FB_SocketCloseAll;
	
	ton_TimeOut: Ton;
	ton_WaitforReconnect: Ton;
	ton_ConnectionEstablised: Ton;
	time_ReconnectTime:TIME:=T#30M;
	byteReceiveString : ARRAY[1..200] OF BYTE;
	FB_BYTE_TO_WORD_1 : FB_CV_BYTE_TO_WORD;
	FB_BYTE_TO_WORD_2 : FB_CV_BYTE_TO_WORD;
	FB_WORD_TO_INT : FB_CV_WORD_TO_INT;
	ton_WaitforNetxtRequest: Ton;
	ton_Wait: Ton;
	int_SuccessCounter: INT;
	int_ReconnectCounter: INT;
	int_ErrorCount: INT;
	fbConvertWordToDword		: FB_CV_WORD_TO_DWORD;			//Convert Word to Dword
	fb_ConvertBytesToLreal		:fb_Convert4BytesToLreal;
	int_SuccessCounterWrite :INT;
	int_NotSuccessCounterWrite :INT;
	i	:INT;
END_VAR


uint_SetPoint_onetenth := LIMIT (0,uint_SetPoint_onetenth,1000);



IF NOT b_Enable THEN			// go to state 0 if not enabled
	i_State := 0;
END_IF


CASE i_State OF
	0:	// wait for enable state
		IF b_Enable THEN
			i_State := 1;
		END_IF
		FB_SocketConnect.bExecute := FALSE;
		FB_SocketSend.bExecute := FALSE;
		FB_SocketSend.bExecute := FALSE;
		ton_TimeOut.IN :=FALSE;	
		ton_ConnectionEstablised.IN := FALSE;
	

	1: // wait, not used now, old state
		i_State := i_State+1;
		
	2: // open socket
		FB_SocketConnect.bExecute := TRUE;
		ton_TimeOut.IN :=TRUE;
		i_State := i_State+1;
		
	3: // wait for connection established	
		IF NOT FB_SocketConnect.bBusy AND NOT FB_SocketConnect.bError THEN
			ton_TimeOut.IN :=FALSE;
			ton_ConnectionEstablised.IN := TRUE;
			i_State := i_State+1;
		ELSIF FB_SocketConnect.bError OR ton_TimeOut.Q THEN
			ton_TimeOut.IN :=FALSE;
			i_State := 100;
		END_IF
	
	4: //connection established, request data
		ton_Wait.IN := TRUE;
		// request FC3, Register 32064, 25 Words --> Real PV Power ff
		byteSendString[1] := 0;
		byteSendString[2] := 1;
		byteSendString[3] := 0;
		byteSendString[4] := 0;
		byteSendString[5] := 0;
		byteSendString[6] := 6;
		byteSendString[7] := LIMIT(1,by_slave_ID,255);			// slave id
		byteSendString[8] := 3;									// function code
		byteSendString[9] := 125;								// adress high
		byteSendString[10] := 64;								// adress low
		byteSendString[11] := 0;								// # of registers high
		byteSendString[12] := 25;								// # of registers low
		
		// clear receive buffer
		FOR i:= 1 TO 200 BY 1 DO
			byteReceiveString[i] := 0;
		END_FOR
		IF ton_Wait.Q THEN
			FB_SocketSend.bExecute := TRUE;
			ton_TimeOut.IN :=TRUE;
			ton_Wait.IN := FALSE;
			i_State := i_State+1;
		END_IF
	
	5: // wait for request sent
		IF NOT FB_SocketSend.bBusy AND NOT FB_SocketSend.bError THEN
			ton_TimeOut.IN :=FALSE;
			FB_SocketSend.bExecute := FALSE;
			i_State := i_State+1;  
		ELSIF FB_SocketSend.bError OR ton_TimeOut.Q THEN
			FB_SocketSend.bExecute := FALSE;
			ton_TimeOut.IN :=FALSE;
			i_State := 100;
		END_IF
		
	6: // wait for data
		ton_Wait.IN := TRUE;
		IF ton_Wait.Q THEN
			FB_SocketReceive.bExecute := TRUE;
			ton_Wait.IN := FALSE;
			i_State := i_State+1; 
		END_IF		 
	
	7:	
		ton_Wait.IN := TRUE;
		IF ton_Wait.Q THEN
			ton_TimeOut.IN :=TRUE;
			i_State := i_State+1; 
		END_IF	
	
	8: // convert received data
		IF NOT FB_SocketReceive.bBusy AND NOT FB_SocketReceive.bError THEN
			int_SuccessCounter := int_SuccessCounter+1;
			ton_TimeOut.IN :=FALSE;
			FB_SocketReceive.bExecute := FALSE;
	
			FB_BYTE_TO_WORD_1(byInputValue_1 := byteReceiveString[14],byInputValue_2 := byteReceiveString[15], Ebyteorderforconvert := Ebyteorder.EBIGENDIAN, woutputvalue => );
			lreal_Voltage_L1L2_V := WORD_TO_LREAL(FB_BYTE_TO_WORD_1.woutputvalue)/10;
			FB_BYTE_TO_WORD_1(byInputValue_1 := byteReceiveString[16],byInputValue_2 := byteReceiveString[17], Ebyteorderforconvert := Ebyteorder.EBIGENDIAN, woutputvalue => );
			lreal_Voltage_L2L3_V := WORD_TO_LREAL(FB_BYTE_TO_WORD_1.woutputvalue)/10;
			FB_BYTE_TO_WORD_1(byInputValue_1 := byteReceiveString[18],byInputValue_2 := byteReceiveString[19], Ebyteorderforconvert := Ebyteorder.EBIGENDIAN, woutputvalue => );
			lreal_Voltage_L3L1_V := WORD_TO_LREAL(FB_BYTE_TO_WORD_1.woutputvalue)/10;
			FB_BYTE_TO_WORD_1(byInputValue_1 := byteReceiveString[20],byInputValue_2 := byteReceiveString[21], Ebyteorderforconvert := Ebyteorder.EBIGENDIAN, woutputvalue => );
			lreal_Voltage_L1_V := WORD_TO_LREAL(FB_BYTE_TO_WORD_1.woutputvalue)/10;
			FB_BYTE_TO_WORD_1(byInputValue_1 := byteReceiveString[22],byInputValue_2 := byteReceiveString[23], Ebyteorderforconvert := Ebyteorder.EBIGENDIAN, woutputvalue => );
			lreal_Voltage_L2_V := WORD_TO_LREAL(FB_BYTE_TO_WORD_1.woutputvalue)/10;
			FB_BYTE_TO_WORD_1(byInputValue_1 := byteReceiveString[24],byInputValue_2 := byteReceiveString[25], Ebyteorderforconvert := Ebyteorder.EBIGENDIAN, woutputvalue => );
			lreal_Voltage_L3_V := WORD_TO_LREAL(FB_BYTE_TO_WORD_1.woutputvalue)/10;


			fb_ConvertBytesToLreal(	by_InputValue_1:= byteReceiveString[10], 
									by_InputValue_2:= byteReceiveString[11], 
									by_InputValue_3:= byteReceiveString[12], 
									by_InputValue_4:= byteReceiveString[13], 
									int_Divider:= 1000, 
									lreal_Output=> );
					
			IF fb_ConvertBytesToLreal.lreal_Output < 100 AND fb_ConvertBytesToLreal.lreal_Output > -1 THEN
				lreal_RealPower_kW := fb_ConvertBytesToLreal.lreal_Output;
			END_IF
			
			fb_ConvertBytesToLreal(	by_InputValue_1:= byteReceiveString[26], 
									by_InputValue_2:= byteReceiveString[27], 
									by_InputValue_3:= byteReceiveString[28], 
									by_InputValue_4:= byteReceiveString[29], 
									int_Divider:= 1000, 
									lreal_Output=> lreal_Current_L1_A);
									
			fb_ConvertBytesToLreal(	by_InputValue_1:= byteReceiveString[30], 
									by_InputValue_2:= byteReceiveString[31], 
									by_InputValue_3:= byteReceiveString[32], 
									by_InputValue_4:= byteReceiveString[33], 
									int_Divider:= 1000, 
									lreal_Output=> lreal_Current_L2_A);

			fb_ConvertBytesToLreal(	by_InputValue_1:= byteReceiveString[34], 
									by_InputValue_2:= byteReceiveString[35], 
									by_InputValue_3:= byteReceiveString[36], 
									by_InputValue_4:= byteReceiveString[37], 
									int_Divider:= 1000, 
									lreal_Output=> lreal_Current_L3_A);
									
			fb_ConvertBytesToLreal(	by_InputValue_1:= byteReceiveString[38], 
									by_InputValue_2:= byteReceiveString[39], 
									by_InputValue_3:= byteReceiveString[40], 
									by_InputValue_4:= byteReceiveString[41], 
									int_Divider:= 1000, 
									lreal_Output=> lreal_PeakPowerDay_kW );

			fb_ConvertBytesToLreal(	by_InputValue_1:= byteReceiveString[42], 
									by_InputValue_2:= byteReceiveString[43], 
									by_InputValue_3:= byteReceiveString[44], 
									by_InputValue_4:= byteReceiveString[45], 
									int_Divider:= 1000, 
									lreal_Output=> lreal_Power2_kW);
			
			fb_ConvertBytesToLreal(	by_InputValue_1:= byteReceiveString[46], 
									by_InputValue_2:= byteReceiveString[47], 
									by_InputValue_3:= byteReceiveString[48], 
									by_InputValue_4:= byteReceiveString[49], 
									int_Divider:= 1000, 
									lreal_Output=>lreal_ReactivePower_kVAr );

			FB_BYTE_TO_WORD_1(byInputValue_1 := byteReceiveString[50],byInputValue_2 := byteReceiveString[51], Ebyteorderforconvert := Ebyteorder.EBIGENDIAN, woutputvalue => );
			lreal_PowerFactor := WORD_TO_LREAL(FB_BYTE_TO_WORD_1.woutputvalue)/1000;
			FB_BYTE_TO_WORD_1(byInputValue_1 := byteReceiveString[52],byInputValue_2 := byteReceiveString[53], Ebyteorderforconvert := Ebyteorder.EBIGENDIAN, woutputvalue => );
			lreal_Frequency_Hz := WORD_TO_LREAL(FB_BYTE_TO_WORD_1.woutputvalue)/100;
			FB_BYTE_TO_WORD_1(byInputValue_1 := byteReceiveString[54],byInputValue_2 := byteReceiveString[55], Ebyteorderforconvert := Ebyteorder.EBIGENDIAN, woutputvalue => );
			lreal_Efficiency := WORD_TO_LREAL(FB_BYTE_TO_WORD_1.woutputvalue)/100;
			FB_BYTE_TO_WORD_1(byInputValue_1 := byteReceiveString[56],byInputValue_2 := byteReceiveString[57], Ebyteorderforconvert := Ebyteorder.EBIGENDIAN, woutputvalue => );
			lreal_InternalTemperature_C := WORD_TO_LREAL(FB_BYTE_TO_WORD_1.woutputvalue)/10;
			FB_BYTE_TO_WORD_1(byInputValue_1 := byteReceiveString[58],byInputValue_2 := byteReceiveString[59], Ebyteorderforconvert := Ebyteorder.EBIGENDIAN, woutputvalue => );
			lreal_IsolationResistance_MOhm := WORD_TO_LREAL(FB_BYTE_TO_WORD_1.woutputvalue)/1000;

		
			//FB_WORD_TO_INT(wInputValue := FB_BYTE_TO_WORD.woutputvalue, iOutputValue => );
			//lreal_RealPower_kW := (INT_TO_LREAL(FB_WORD_TO_INT.iOutputValue))/1000;

			i_State := i_State+1;
		ELSIF FB_SocketSend.bError OR ton_TimeOut.Q THEN
 			FB_SocketReceive.bExecute := FALSE;
			ton_TimeOut.IN :=FALSE;
			i_State := 100;
		END_IF
	
	9: // for for next request
		ton_WaitforNetxtRequest.IN := TRUE;
		IF NOT b_Enable THEN
			ton_WaitforNetxtRequest.IN := FALSE;
			i_State := 50;
		END_IF
		IF ton_WaitforNetxtRequest.Q THEN
			ton_WaitforNetxtRequest.IN := FALSE;
			i_State := 20;
		END_IF
		IF 	ton_ConnectionEstablised.Q THEN 
			ton_WaitforNetxtRequest.IN := FALSE;
			i_State := 50;
		END_IF

	20: // write Setpoint
		ton_Wait.IN := TRUE;
		// request FC6 write register, Register 40125, 2 Word power setpoint
		byteSendString[1] := 0;
		byteSendString[2] := 1;
		byteSendString[3] := 0;
		byteSendString[4] := 0;
		byteSendString[5] := 0;
		byteSendString[6] := 6;
		byteSendString[7] := LIMIT(1,by_slave_ID,255);			// slave id
		byteSendString[8] := 6;									// function code
		byteSendString[9] := 156;								// adress high
		byteSendString[10] := 189;								// adress low
		byteSendString[11] := WORD_TO_BYTE(SHR(UINT_TO_WORD(uint_SetPoint_onetenth),8) AND 16#FFFF);		// # Value high
		byteSendString[12] := WORD_TO_BYTE(UINT_TO_WORD(uint_SetPoint_onetenth) AND 16#FFFF);				// # Value low		
	// clear receive buffer
		FOR i:= 1 TO 200 BY 1 DO
			byteReceiveString[i] := 0;
		END_FOR		
		IF ton_Wait.Q THEN
			FB_SocketSend.bExecute := TRUE;
			ton_TimeOut.IN :=TRUE;
			ton_Wait.IN := FALSE;
			i_State := i_State+1;
		END_IF
	
	21: // wait for request sent
		IF NOT FB_SocketSend.bBusy AND NOT FB_SocketSend.bError THEN
			ton_TimeOut.IN :=FALSE;
			FB_SocketSend.bExecute := FALSE;
			i_State := i_State+1;  
		ELSIF FB_SocketSend.bError OR ton_TimeOut.Q THEN
			FB_SocketSend.bExecute := FALSE;
			ton_TimeOut.IN :=FALSE;
			i_State := 100;
		END_IF		
		
	22: // wait for data
		ton_Wait.IN := TRUE;
		IF ton_Wait.Q THEN
			FB_SocketReceive.bExecute := TRUE;
			ton_Wait.IN := FALSE;
			i_State := i_State+1; 
		END_IF		 
	
	23:	
		ton_Wait.IN := TRUE;
		IF ton_Wait.Q THEN
			ton_TimeOut.IN :=TRUE;
			i_State := i_State+1; 
		END_IF	
	
	24: // Verify received data / writing succesful
		IF NOT FB_SocketReceive.bBusy AND NOT FB_SocketReceive.bError THEN
			
			IF 	byteReceiveString[5] = byteSendString[5] AND
				byteReceiveString[6] = byteSendString[6] AND
				byteReceiveString[7] = byteSendString[7] AND
				byteReceiveString[8] = byteSendString[8] AND 
				byteReceiveString[9] = byteSendString[9] AND
				byteReceiveString[10] = byteSendString[10] THEN
				int_SuccessCounterWrite := int_SuccessCounterWrite+1;
			ELSE
				int_NotSuccessCounterWrite := int_NotSuccessCounterWrite+1;
			END_IF
		

			i_State := i_State+1;
		ELSIF FB_SocketSend.bError OR ton_TimeOut.Q THEN
 			int_NotSuccessCounterWrite := int_NotSuccessCounterWrite+1;
			FB_SocketReceive.bExecute := FALSE;
			ton_TimeOut.IN :=FALSE;
			i_State := 100;
		END_IF
	
	25: // for for next request
		ton_WaitforNetxtRequest.IN := TRUE;
		IF NOT b_Enable THEN
			ton_WaitforNetxtRequest.IN := FALSE;
			i_State := 50;
		END_IF
		IF ton_WaitforNetxtRequest.Q THEN
			ton_WaitforNetxtRequest.IN := FALSE;
			i_State := 4;
		END_IF
		IF 	ton_ConnectionEstablised.Q THEN 
			ton_WaitforNetxtRequest.IN := FALSE;
			i_State := 50;
		END_IF	
		
		
	50: // close sockets
		FB_CloseSockets.bExecute := TRUE;
		ton_TimeOut.IN :=TRUE;
		i_State := i_State+1;
		
	51: // wait for sockets closed
		
		IF NOT FB_CloseSockets.bBusy THEN
			int_ReconnectCounter := int_ReconnectCounter+1;
			FB_CloseSockets.bExecute := FALSE;
			i_State := 0;
		ELSIF FB_CloseSockets.bError THEN
			int_ReconnectCounter := int_ReconnectCounter+1;
			FB_CloseSockets.bExecute := FALSE;
			i_State := 0;
		END_IF



		
		
		
		
		
		
	100: // wait state for reconect
		
		FB_SocketConnect.bExecute := FALSE;
		FB_SocketSend.bExecute := FALSE;
		FB_SocketReceive.bExecute := FALSE;
		ton_ConnectionEstablised.IN := FALSE;
		ton_TimeOut.IN :=FALSE;
		ton_WaitforReconnect.IN := TRUE;
		IF ton_WaitforReconnect.Q THEN
			int_ErrorCount := int_ErrorCount+1;
			ton_WaitforReconnect.IN := FALSE;
			i_State := 50;
		END_IF
	
END_CASE



FB_SocketConnect(
	sSrvNetId := '',
	sRemoteHost := str_IPAdress,
	nRemotePort := 502,
	bExecute := ,
	tTimeout := T#1S,
	bBusy =>,
	bError =>,
	nErrId =>,
	hSocket => hSocket);
	
FB_SocketSend(
	sSrvNetId:= '', 
	hSocket:= hSocket, 
	cbLen:= 12,
	pSrc:= ADR( byteSendString ), 
	bExecute:= , 
	tTimeout:= T#3S, 
	bBusy=> , 
	bError=> , 
	nErrId=> );
	
FB_SocketReceive(
	sSrvNetId:= '', 
	hSocket:= hSocket, 
	cbLen:= 200, 
	pDest:= ADR( byteReceiveString ), 
	bExecute:= , 
	tTimeout:= T#3S, 
	bBusy=> , 
	bError=> , 
	nErrId=> , 
	nRecBytes=> );

FB_CloseSockets(
	sSrvNetId:= '', 
	bExecute:= , 
	tTimeout:= T#2S, 
	bBusy=> , 
	bError=> , 
	nErrId=> );
	
ton_TimeOut(PT := T#5S);
ton_WaitforReconnect(PT := T#10S);
ton_ConnectionEstablised(pt := time_ReconnectTime);
ton_WaitforNetxtRequest(PT:= T#2S);
ton_Wait(PT:=T#2S);

END_FUNCTION_BLOCK

// ---- FB/fb_Convert4BytesToLreal.TcPOU
FUNCTION_BLOCK fb_Convert4BytesToLreal
VAR_INPUT
	by_InputValue_1:BYTE;
	by_InputValue_2:BYTE;
	by_InputValue_3:BYTE;
	by_InputValue_4:BYTE;
	int_Divider: INT;
END_VAR
VAR_OUTPUT
	lreal_Output:LREAL;
END_VAR
VAR
	FB_BYTE_TO_WORD_1 : FB_CV_BYTE_TO_WORD;
	FB_BYTE_TO_WORD_2 : FB_CV_BYTE_TO_WORD;
	fbConvertWordToDword		: FB_CV_WORD_TO_DWORD;			//Convert Word to Dword

END_VAR

IF int_Divider =0 THEN
	int_Divider :=1;
END_IF
FB_BYTE_TO_WORD_1(byInputValue_1 := by_InputValue_1,byInputValue_2 := by_InputValue_2, Ebyteorderforconvert := Ebyteorder.ebigENDIAN, woutputvalue => );
FB_BYTE_TO_WORD_2(byInputValue_1 := by_InputValue_3,byInputValue_2 := by_InputValue_4, Ebyteorderforconvert := Ebyteorder.ebigENDIAN, woutputvalue => );

fbConvertWordToDword(wInputValue_1:= FB_BYTE_TO_WORD_1.woutputvalue, wInputValue_2:= FB_BYTE_TO_WORD_2.woutputvalue, eByteOrderForConvert:= eByteOrder.eBigEndian , dwOutputValue=> );
lreal_Output :=DINT_TO_LREAL( DWORD_TO_DINT(fbConvertWordToDword.dwOutputValue))/int_Divider;

END_FUNCTION_BLOCK

// ---- POUs/prgPV_separate.TcPOU
PROGRAM prgPV_separate
VAR
	fbPVCounter_1			: FB_EnergyCounter;
	fbPVCounter_2			: FB_EnergyCounter;
	lrPowerPV				: LREAL;				
		// extend or reduce amount of PV Inverters
	lrPowerPV_1				: LREAL;				
	lrPowerPV_2				: LREAL;				

	str_IP: STRING(15) := '172.16.127.240';
	FB_PV_1:FB_TCPModbusRequest_PV_Huawei_inclWrite_oneTurn;	

	fb_Meter_1		: FB_EM_Electric_3P_Ext_Input;
	fbPVInt_1		: FB_PV_Power;
	fb_Meter_2		: FB_EM_Electric_3P_Ext_Input;
	fbPVInt_2		: FB_PV_Power;
	

	FB_PID_Inverter :FB_PID;

	uint_setPoint_onetenth: UINT;					

	rPValue: REAL := 0.05;
	udint_IValue: UDINT:=250;
	udint_DValue: UDINT:=30;

	unit_Temp: UINT;
	real_max: REAL:=1000;
	real_min: REAL:=10;

	int_state: INT;
	ton_State_Timeout: TON;
	mtest: BOOL:=TRUE;
END_VAR
VAR PERSISTENT
	lrCounterPV_1				: LREAL;			
	lrCounterPV_2				: LREAL;				
	m_Direction: BOOL:= TRUE;
END_VAR

// state maschine for talking to each PV inverter by the time

CASE int_state OF
	0: // wait state
		int_state := 10;
		FB_PV_1.b_Enable := FALSE;
		
	10: //talk to first PV
		IF FB_PV_1.i_State = 0 THEN
			int_state := int_state+1;
		END_IF
	
	11: // start first poll
		FB_PV_1.b_Enable := TRUE;
		FB_PV_1.by_slave_ID:= 1;
		ton_State_Timeout.IN := TRUE;
		IF FB_PV_1.i_State <> 0 THEN
			int_state := int_state+1;
		END_IF
 
		
	12: // wait for data received
		FB_PV_1.b_Enable := FALSE;
		IF FB_PV_1.i_State = 0 AND NOT FB_PV_1.FB_SocketReceive.bError THEN
 			lrPowerPV_1 := FB_PV_1.lreal_RealPower_kW;
			ton_State_Timeout.IN := FALSE;
			int_state := int_state+1;
		ELSIF ton_State_Timeout.Q THEN
			ton_State_Timeout.IN := FALSE;
			int_state := int_state+1;
		END_IF
		
	13: // go to next poll
		int_state := 20;
		
	20: //talk to second PV
		IF FB_PV_1.i_State = 0 THEN
			int_state := int_state+1;
		END_IF
	
	21: // start first poll
		FB_PV_1.b_Enable := TRUE;
		FB_PV_1.by_slave_ID:= 2;
		ton_State_Timeout.IN := TRUE;
		IF FB_PV_1.i_State <> 0 THEN
			int_state := int_state+1;
		END_IF
 
		
	22: // wait for data received
		FB_PV_1.b_Enable := FALSE;
		IF FB_PV_1.i_State = 0 AND NOT FB_PV_1.FB_SocketReceive.bError THEN
 			lrPowerPV_2 := FB_PV_1.lreal_RealPower_kW;
			ton_State_Timeout.IN := FALSE;
			int_state := int_state+1;
		ELSIF ton_State_Timeout.Q THEN
			ton_State_Timeout.IN := FALSE;
			int_state := int_state+1;
		END_IF		
	23: // go to next poll
		int_state := 0;		
		
END_CASE
ton_State_Timeout(pt:= T#1M);



		
FB_PV_1(
	b_Enable:= , 
	by_slave_ID:= , 
	str_IPAdress:= str_ip, 
	uint_SetPoint_onetenth:= uint_setPoint_onetenth, 
	lreal_RealPower_kW=> ,  );


	

fbPVCounter_1(	byActiveTariff := 1,	
				lrPowerInput := 0-lrPowerPV_1,
				lrTotalCounterEnergy_Production => lrCounterPV_1);

fbPVCounter_2(	byActiveTariff := 1,	
				lrPowerInput := 0-lrPowerPV_2,
				lrTotalCounterEnergy_Production => lrCounterPV_2);

lrPowerPV := lrPowerPV_1 + lrPowerPV_2;

fbPVInt_1(
	bEnable:= TRUE, 
	bPowerDataInvers:= , 
	diNrOfEM_IN_PV:= fb_Meter_1.diNrOfEM_OUT, 
	stDataPv=> , 
	diNrOfPv_OUT=> );
	
fb_Meter_1(
	bEnable:= TRUE, 
	bPowerDataInvers:= , 
	bErrorExt:= , 
	bWarningExt:= , 
	lrTotalCounterEnergy_Consumption:= , 
	lrTotalCounterEnergy_Production:= , 
	lrCounterEnergyT1_Consumption:= , 
	lrCounterEnergyT2_Consumption:= , 
	lrCounterEnergyT1_Production:= , 
	lrCounterEnergyT2_Production:= , 
	lrCurrentL1:= , 
	lrVoltageL1N:= , 
	lrVoltageL1L2:= , 
	lrPowerL1:= , 
	lrCurrentL2:= , 
	lrVoltageL2N:= , 
	lrVoltageL2L3:= , 
	lrPowerL2:= , 
	lrCurrentL3:= , 
	lrVoltageL3N:= , 
	lrVoltageL3L1:= , 
	lrPowerL3:= , 
	lrPowerTotal:= lrPowerPV_1,
	lrFrequency:= , 
	lrReactivePowerTotal:= , 
	lrApparentPowerTotal:= , 
	stDataEMPower=> , 
	stDataEMCounter=> , 
	diNrOfEM_OUT=> );

	

fbPVInt_2(
	bEnable:= TRUE, 
	bPowerDataInvers:= , 
	diNrOfEM_IN_PV:= fb_Meter_2.diNrOfEM_OUT, 
	stDataPv=> , 
	diNrOfPv_OUT=> );
	
fb_Meter_2(	
	bEnable:= TRUE, 
	bPowerDataInvers:= , 
	bErrorExt:= , 
	bWarningExt:= , 
	lrTotalCounterEnergy_Consumption:= , 
	lrTotalCounterEnergy_Production:= , 
	lrCounterEnergyT1_Consumption:= , 
	lrCounterEnergyT2_Consumption:= , 
	lrCounterEnergyT1_Production:= , 
	lrCounterEnergyT2_Production:= , 
	lrCurrentL1:= , 
	lrVoltageL1N:= , 
	lrVoltageL1L2:= , 
	lrPowerL1:= , 
	lrCurrentL2:= , 
	lrVoltageL2N:= , 
	lrVoltageL2L3:= , 
	lrPowerL2:= , 
	lrCurrentL3:= , 
	lrVoltageL3N:= , 
	lrVoltageL3L1:= , 
	lrPowerL3:= , 
	lrPowerTotal:= lrPowerPV_2,
	lrFrequency:= , 
	lrReactivePowerTotal:= , 
	lrApparentPowerTotal:= , 
	stDataEMPower=> , 
	stDataEMCounter=> , 
	diNrOfEM_OUT=> );

	
FB_PID_Inverter(
		bEnable:= TRUE, 
		rSetpoint:= -LIMIT(0,prgGrid.rSizeGridDelivery,30), 
		udiIValue:= udint_IValue, 
		udiDValue:= udint_DValue, 
		udiDamping:= 0, 
		rPValue:= rPValue, 
		rMaxValue:= real_max, 
		rMinValue:= real_min, 
		rNeutralZone:= 1, 
		bDirection:= m_Direction, 
		rActualValue:=  LREAL_TO_REAL(prgGrid.fbEM1.stDataEMPowerRealTime.lrPowerTotal),
		rQController=> );
IF mtest THEN
	uint_setPoint_onetenth := REAL_TO_UINT(FB_PID_Inverter.rQController);
END_IF

END_PROGRAM

// ---- FB/FB_TCPModbusRequest_PV_Huawei_inclWrite_oneTurn.TcPOU
FUNCTION_BLOCK FB_TCPModbusRequest_PV_Huawei_inclWrite_oneTurn
VAR_INPUT
	b_Enable: BOOL;
	by_slave_ID	:BYTE;
	str_IPAdress: STRING(15);
	uint_SetPoint_onetenth	:UINT;
END_VAR
VAR_OUTPUT

	lreal_RealPower_kW:LREAL;
	lreal_Voltage_L1L2_V: LREAL;
	lreal_Voltage_L2L3_V: LREAL;
	lreal_Voltage_L3L1_V: LREAL;
	lreal_Voltage_L1_V: LREAL;
	lreal_Voltage_L2_V: LREAL;
	lreal_Voltage_L3_V: LREAL;
	lreal_Current_L1_A: LREAL;
	lreal_Current_L2_A: LREAL;
	lreal_Current_L3_A: LREAL;
	lreal_PeakPowerDay_kW: LREAL;
	lreal_Power2_kW: LREAL;
	lreal_ReactivePower_kVAr: LREAL;
	lreal_PowerFactor: LREAL;
	lreal_Frequency_Hz: LREAL;
	lreal_Efficiency: LREAL;
	lreal_InternalTemperature_C: LREAL;
	lreal_IsolationResistance_MOhm: LREAL;
END_VAR
VAR
	i_State:INT;
	FB_SocketConnect : FB_SocketConnect;
	hSocket : T_HSOCKET;
	FB_SocketSend : FB_SocketSend;
	FB_SocketReceive : FB_SocketReceive;
	byteSendString : ARRAY[1..12] OF BYTE;
	FB_CloseSockets: FB_SocketCloseAll;
	
	ton_TimeOut: Ton;
	ton_WaitforReconnect: Ton;
	ton_ConnectionEstablised: Ton;
	time_ReconnectTime:TIME:=T#30M;
	byteReceiveString : ARRAY[1..200] OF BYTE;
	FB_BYTE_TO_WORD_1 : FB_CV_BYTE_TO_WORD;
	FB_BYTE_TO_WORD_2 : FB_CV_BYTE_TO_WORD;
	FB_WORD_TO_INT : FB_CV_WORD_TO_INT;
	ton_WaitforNetxtRequest: Ton;
	ton_Wait: Ton;
	int_SuccessCounter: INT;
	int_ReconnectCounter: INT;
	int_ErrorCount: INT;
	fbConvertWordToDword		: FB_CV_WORD_TO_DWORD;			//Convert Word to Dword
	fb_ConvertBytesToLreal		:fb_Convert4BytesToLreal;
	int_SuccessCounterWrite :INT;
	int_NotSuccessCounterWrite :INT;
	i	:INT;
	r_trig_Enable: R_trig;
	int_count: int;
	i_State_temp: INT;
	f_trig_Busy: f_trig;
	time_wait: TIME:= T#3S;
END_VAR


uint_SetPoint_onetenth := LIMIT (0,uint_SetPoint_onetenth,1000);



r_trig_Enable( clk := b_Enable);

CASE i_State OF
	0:	// wait for enable rising edge
		IF r_trig_Enable.Q THEN
			i_State := 1;
		END_IF
		FB_SocketConnect.bExecute := FALSE;
		FB_SocketSend.bExecute := FALSE;
		FB_SocketSend.bExecute := FALSE;
		ton_TimeOut.IN :=FALSE;	
		ton_ConnectionEstablised.IN := FALSE;
	

	1: // wait, not used now, old state
		i_State := i_State+1;
		
	2: // open socket
		FB_SocketConnect.bExecute := TRUE;
		ton_TimeOut.IN :=TRUE;
		i_State := i_State+1;
		
	3: // wait for connection established	
		IF NOT FB_SocketConnect.bBusy AND NOT FB_SocketConnect.bError THEN
			ton_TimeOut.IN :=FALSE;
			ton_ConnectionEstablised.IN := TRUE;
			i_State := i_State+1;
		ELSIF FB_SocketConnect.bError OR ton_TimeOut.Q THEN
			ton_TimeOut.IN :=FALSE;
			i_State := 100;
		END_IF
	
	4: //connection established, request data
		ton_Wait.IN := TRUE;
		// request FC3, Register 32064, 25 Words --> Real PV Power ff
		byteSendString[1] := 0;
		byteSendString[2] := 1;
		byteSendString[3] := 0;
		byteSendString[4] := 0;
		byteSendString[5] := 0;
		byteSendString[6] := 6;
		byteSendString[7] := LIMIT(1,by_slave_ID,255);			// slave id
		byteSendString[8] := 3;									// function code
		byteSendString[9] := 125;								// adress high
		byteSendString[10] := 64;								// adress low
		byteSendString[11] := 0;								// # of registers high
		byteSendString[12] := 25;								// # of registers low
		
		// clear receive buffer
		FOR i:= 1 TO 200 BY 1 DO
			byteReceiveString[i] := 0;
		END_FOR
		IF ton_Wait.Q THEN
			FB_SocketSend.bExecute := TRUE;
			ton_TimeOut.IN :=TRUE;
			ton_Wait.IN := FALSE;
			i_State := i_State+1;
		END_IF
	
	5: // wait for request sent
		IF NOT FB_SocketSend.bBusy AND NOT FB_SocketSend.bError THEN
			ton_TimeOut.IN :=FALSE;
			FB_SocketSend.bExecute := FALSE;
			i_State := i_State+1;  
		ELSIF FB_SocketSend.bError OR ton_TimeOut.Q THEN
			FB_SocketSend.bExecute := FALSE;
			ton_TimeOut.IN :=FALSE;
			i_State := 100;
		END_IF
		
	6: // wait for data
		ton_Wait.IN := TRUE;
		IF ton_Wait.Q THEN
			FB_SocketReceive.bExecute := TRUE;
			ton_Wait.IN := FALSE;
			i_State := i_State+1; 
		END_IF		 
	
	7:	
		ton_TimeOut.IN :=TRUE;
		IF f_trig_Busy.Q THEN
			FB_SocketReceive.bExecute := FALSE;
			i_State := i_State+1; 
		END_IF	
		IF ton_TimeOut.Q THEN
			FB_SocketReceive.bExecute := FALSE;
			ton_TimeOut.IN :=FALSE;
			i_State := 100;			
		END_IF
	
	8: // convert received data
		IF NOT FB_SocketReceive.bBusy AND NOT FB_SocketReceive.bError AND FB_SocketReceive.nRecBytes <> 0 THEN 
			int_SuccessCounter := int_SuccessCounter+1;
			ton_TimeOut.IN :=FALSE;
			FB_SocketReceive.bExecute := FALSE;
	
			FB_BYTE_TO_WORD_1(byInputValue_1 := byteReceiveString[14],byInputValue_2 := byteReceiveString[15], Ebyteorderforconvert := Ebyteorder.EBIGENDIAN, woutputvalue => );
			lreal_Voltage_L1L2_V := WORD_TO_LREAL(FB_BYTE_TO_WORD_1.woutputvalue)/10;
			FB_BYTE_TO_WORD_1(byInputValue_1 := byteReceiveString[16],byInputValue_2 := byteReceiveString[17], Ebyteorderforconvert := Ebyteorder.EBIGENDIAN, woutputvalue => );
			lreal_Voltage_L2L3_V := WORD_TO_LREAL(FB_BYTE_TO_WORD_1.woutputvalue)/10;
			FB_BYTE_TO_WORD_1(byInputValue_1 := byteReceiveString[18],byInputValue_2 := byteReceiveString[19], Ebyteorderforconvert := Ebyteorder.EBIGENDIAN, woutputvalue => );
			lreal_Voltage_L3L1_V := WORD_TO_LREAL(FB_BYTE_TO_WORD_1.woutputvalue)/10;
			FB_BYTE_TO_WORD_1(byInputValue_1 := byteReceiveString[20],byInputValue_2 := byteReceiveString[21], Ebyteorderforconvert := Ebyteorder.EBIGENDIAN, woutputvalue => );
			lreal_Voltage_L1_V := WORD_TO_LREAL(FB_BYTE_TO_WORD_1.woutputvalue)/10;
			FB_BYTE_TO_WORD_1(byInputValue_1 := byteReceiveString[22],byInputValue_2 := byteReceiveString[23], Ebyteorderforconvert := Ebyteorder.EBIGENDIAN, woutputvalue => );
			lreal_Voltage_L2_V := WORD_TO_LREAL(FB_BYTE_TO_WORD_1.woutputvalue)/10;
			FB_BYTE_TO_WORD_1(byInputValue_1 := byteReceiveString[24],byInputValue_2 := byteReceiveString[25], Ebyteorderforconvert := Ebyteorder.EBIGENDIAN, woutputvalue => );
			lreal_Voltage_L3_V := WORD_TO_LREAL(FB_BYTE_TO_WORD_1.woutputvalue)/10;


			fb_ConvertBytesToLreal(	by_InputValue_1:= byteReceiveString[10], 
									by_InputValue_2:= byteReceiveString[11], 
									by_InputValue_3:= byteReceiveString[12], 
									by_InputValue_4:= byteReceiveString[13], 
									int_Divider:= 1000, 
									lreal_Output=> );
					
			IF fb_ConvertBytesToLreal.lreal_Output < 100 AND fb_ConvertBytesToLreal.lreal_Output > -1 THEN
				lreal_RealPower_kW := fb_ConvertBytesToLreal.lreal_Output;
			END_IF
			
			fb_ConvertBytesToLreal(	by_InputValue_1:= byteReceiveString[26], 
									by_InputValue_2:= byteReceiveString[27], 
									by_InputValue_3:= byteReceiveString[28], 
									by_InputValue_4:= byteReceiveString[29], 
									int_Divider:= 1000, 
									lreal_Output=> lreal_Current_L1_A);
									
			fb_ConvertBytesToLreal(	by_InputValue_1:= byteReceiveString[30], 
									by_InputValue_2:= byteReceiveString[31], 
									by_InputValue_3:= byteReceiveString[32], 
									by_InputValue_4:= byteReceiveString[33], 
									int_Divider:= 1000, 
									lreal_Output=> lreal_Current_L2_A);

			fb_ConvertBytesToLreal(	by_InputValue_1:= byteReceiveString[34], 
									by_InputValue_2:= byteReceiveString[35], 
									by_InputValue_3:= byteReceiveString[36], 
									by_InputValue_4:= byteReceiveString[37], 
									int_Divider:= 1000, 
									lreal_Output=> lreal_Current_L3_A);
									
			fb_ConvertBytesToLreal(	by_InputValue_1:= byteReceiveString[38], 
									by_InputValue_2:= byteReceiveString[39], 
									by_InputValue_3:= byteReceiveString[40], 
									by_InputValue_4:= byteReceiveString[41], 
									int_Divider:= 1000, 
									lreal_Output=> lreal_PeakPowerDay_kW );

			fb_ConvertBytesToLreal(	by_InputValue_1:= byteReceiveString[42], 
									by_InputValue_2:= byteReceiveString[43], 
									by_InputValue_3:= byteReceiveString[44], 
									by_InputValue_4:= byteReceiveString[45], 
									int_Divider:= 1000, 
									lreal_Output=> lreal_Power2_kW);
			
			fb_ConvertBytesToLreal(	by_InputValue_1:= byteReceiveString[46], 
									by_InputValue_2:= byteReceiveString[47], 
									by_InputValue_3:= byteReceiveString[48], 
									by_InputValue_4:= byteReceiveString[49], 
									int_Divider:= 1000, 
									lreal_Output=>lreal_ReactivePower_kVAr );

			FB_BYTE_TO_WORD_1(byInputValue_1 := byteReceiveString[50],byInputValue_2 := byteReceiveString[51], Ebyteorderforconvert := Ebyteorder.EBIGENDIAN, woutputvalue => );
			lreal_PowerFactor := WORD_TO_LREAL(FB_BYTE_TO_WORD_1.woutputvalue)/1000;
			FB_BYTE_TO_WORD_1(byInputValue_1 := byteReceiveString[52],byInputValue_2 := byteReceiveString[53], Ebyteorderforconvert := Ebyteorder.EBIGENDIAN, woutputvalue => );
			lreal_Frequency_Hz := WORD_TO_LREAL(FB_BYTE_TO_WORD_1.woutputvalue)/100;
			FB_BYTE_TO_WORD_1(byInputValue_1 := byteReceiveString[54],byInputValue_2 := byteReceiveString[55], Ebyteorderforconvert := Ebyteorder.EBIGENDIAN, woutputvalue => );
			lreal_Efficiency := WORD_TO_LREAL(FB_BYTE_TO_WORD_1.woutputvalue)/100;
			FB_BYTE_TO_WORD_1(byInputValue_1 := byteReceiveString[56],byInputValue_2 := byteReceiveString[57], Ebyteorderforconvert := Ebyteorder.EBIGENDIAN, woutputvalue => );
			lreal_InternalTemperature_C := WORD_TO_LREAL(FB_BYTE_TO_WORD_1.woutputvalue)/10;
			FB_BYTE_TO_WORD_1(byInputValue_1 := byteReceiveString[58],byInputValue_2 := byteReceiveString[59], Ebyteorderforconvert := Ebyteorder.EBIGENDIAN, woutputvalue => );
			lreal_IsolationResistance_MOhm := WORD_TO_LREAL(FB_BYTE_TO_WORD_1.woutputvalue)/1000;

		
			//FB_WORD_TO_INT(wInputValue := FB_BYTE_TO_WORD.woutputvalue, iOutputValue => );
			//lreal_RealPower_kW := (INT_TO_LREAL(FB_WORD_TO_INT.iOutputValue))/1000;
			int_count := 0;
			i_State := i_State+1;
		ELSIF FB_SocketReceive.nRecBytes = 0 THEN
			
			IF int_count > 5 THEN
			 	i_State := 100;
				int_count := 0;
			ELSE
				i_State := 4;
				int_count := int_count + 1;
			END_IF	

(*		ELSIF FB_SocketSend.bError OR ton_TimeOut.Q THEN
 			FB_SocketReceive.bExecute := FALSE;
			ton_TimeOut.IN :=FALSE;
			i_State := 100;
*)		END_IF
	
	9: // for for next request
		IF FB_SocketReceive.nRecBytes = 0 THEN 
			i_State := 4;
		END_IF
		ton_WaitforNetxtRequest.IN := TRUE;
		IF ton_WaitforNetxtRequest.Q THEN
			ton_WaitforNetxtRequest.IN := FALSE;
			i_State := 20;
		END_IF
		IF 	ton_ConnectionEstablised.Q THEN 
			ton_WaitforNetxtRequest.IN := FALSE;
			i_State := 50;
		END_IF

	20: // write Setpoint
		ton_Wait.IN := TRUE;
		// request FC6 write register, Register 40125, 2 Word power setpoint
		byteSendString[1] := 0;
		byteSendString[2] := 1;
		byteSendString[3] := 0;
		byteSendString[4] := 0;
		byteSendString[5] := 0;
		byteSendString[6] := 6;
		byteSendString[7] := LIMIT(1,by_slave_ID,255);			// slave id
		byteSendString[8] := 6;									// function code
		byteSendString[9] := 156;								// adress high
		byteSendString[10] := 189;								// adress low
		byteSendString[11] := WORD_TO_BYTE(SHR(UINT_TO_WORD(uint_SetPoint_onetenth),8) AND 16#FFFF);		// # Value high
		byteSendString[12] := WORD_TO_BYTE(UINT_TO_WORD(uint_SetPoint_onetenth) AND 16#FFFF);				// # Value low		
	// clear receive buffer
		FOR i:= 1 TO 200 BY 1 DO
			byteReceiveString[i] := 0;
		END_FOR		
		IF ton_Wait.Q THEN
			FB_SocketSend.bExecute := TRUE;
			ton_TimeOut.IN :=TRUE;
			ton_Wait.IN := FALSE;
			i_State := i_State+1;
		END_IF
	
	21: // wait for request sent
		IF NOT FB_SocketSend.bBusy AND NOT FB_SocketSend.bError THEN
			ton_TimeOut.IN :=FALSE;
			FB_SocketSend.bExecute := FALSE;
			i_State := i_State+1;  
		ELSIF FB_SocketSend.bError OR ton_TimeOut.Q THEN
			FB_SocketSend.bExecute := FALSE;
			ton_TimeOut.IN :=FALSE;
			i_State := 100;
		END_IF		
		
	22: // wait for data
		ton_Wait.IN := TRUE;
		IF ton_Wait.Q THEN
			FB_SocketReceive.bExecute := TRUE;
			ton_Wait.IN := FALSE;
			i_State := i_State+1; 
		END_IF		 
	
	23:	
		ton_Wait.IN := TRUE;
		IF ton_Wait.Q THEN
			ton_TimeOut.IN :=TRUE;
			i_State := i_State+1; 
		END_IF	
	
	24: // Verify received data / writing succesful
		 	FB_SocketReceive.bExecute := FALSE;
		IF NOT FB_SocketReceive.bBusy AND NOT FB_SocketReceive.bError THEN
			
			IF 	byteReceiveString[5] = byteSendString[5] AND
				byteReceiveString[6] = byteSendString[6] AND
				byteReceiveString[7] = byteSendString[7] AND
				byteReceiveString[8] = byteSendString[8] AND 
				byteReceiveString[9] = byteSendString[9] AND
				byteReceiveString[10] = byteSendString[10] THEN
				int_SuccessCounterWrite := int_SuccessCounterWrite+1;
				i_State := i_State+1;
				int_count := 0;
			ELSE
				int_NotSuccessCounterWrite := int_NotSuccessCounterWrite+1;
				IF int_count > 5 THEN
				 	i_State := 100;
					int_count := 0;
				ELSE
					i_State := 20;
					int_count := int_count + 1;
				END_IF	
			END_IF
		

			
		ELSIF FB_SocketSend.bError OR ton_TimeOut.Q THEN
 			int_NotSuccessCounterWrite := int_NotSuccessCounterWrite+1;
			FB_SocketReceive.bExecute := FALSE;
			ton_TimeOut.IN :=FALSE;
			i_State := 100;
		END_IF
	
	25: // for for next request
		ton_WaitforNetxtRequest.IN := TRUE;
		IF ton_WaitforNetxtRequest.Q THEN
			ton_WaitforNetxtRequest.IN := FALSE;
			i_State := 50;
		END_IF
		IF 	ton_ConnectionEstablised.Q THEN 
			ton_WaitforNetxtRequest.IN := FALSE;
			i_State := 50;
		END_IF	
		
		
	50: // close sockets
		FB_CloseSockets.bExecute := TRUE;
		ton_TimeOut.IN :=TRUE;
		i_State := i_State+1;
		
	51: // wait for sockets closed
		
		IF NOT FB_CloseSockets.bBusy THEN
			int_ReconnectCounter := int_ReconnectCounter+1;
			FB_CloseSockets.bExecute := FALSE;
			i_State := 0;
		ELSIF FB_CloseSockets.bError THEN
			int_ReconnectCounter := int_ReconnectCounter+1;
			FB_CloseSockets.bExecute := FALSE;
			i_State := 0;
		END_IF

	100: // wait state for reconect
		
		FB_SocketConnect.bExecute := FALSE;
		FB_SocketSend.bExecute := FALSE;
		FB_SocketReceive.bExecute := FALSE;
		ton_ConnectionEstablised.IN := FALSE;
		ton_TimeOut.IN :=FALSE;
		ton_WaitforReconnect.IN := TRUE;
		IF ton_WaitforReconnect.Q THEN
			int_ErrorCount := int_ErrorCount+1;
			ton_WaitforReconnect.IN := FALSE;
			i_State := 50;
		END_IF
	
END_CASE
f_trig_Busy(clk := FB_SocketReceive.bBusy);


FB_SocketConnect(
	sSrvNetId := '',
	sRemoteHost := str_IPAdress,
	nRemotePort := 502,
	bExecute := ,
	tTimeout := T#5S,
	bBusy =>,
	bError =>,
	nErrId =>,
	hSocket => hSocket);
	
FB_SocketSend(
	sSrvNetId:= '', 
	hSocket:= hSocket, 
	cbLen:= 12,
	pSrc:= ADR( byteSendString ), 
	bExecute:= , 
	tTimeout:= T#5S, 
	bBusy=> , 
	bError=> , 
	nErrId=> );
	
FB_SocketReceive(
	sSrvNetId:= '', 
	hSocket:= hSocket, 
	cbLen:= 200, 
	pDest:= ADR( byteReceiveString ), 
	bExecute:= , 
	tTimeout:= T#5S, 
	bBusy=> , 
	bError=> , 
	nErrId=> , 
	nRecBytes=> );

FB_CloseSockets(
	sSrvNetId:= '', 
	bExecute:= , 
	tTimeout:= T#2S, 
	bBusy=> , 
	bError=> , 
	nErrId=> );
	
ton_TimeOut(PT := T#10S);
ton_WaitforReconnect(PT := T#10S);
ton_ConnectionEstablised(pt := time_ReconnectTime);
ton_WaitforNetxtRequest(PT:= T#2S);
ton_Wait(PT:=time_wait);

END_FUNCTION_BLOCK

// ---- POUs/prgBattery.TcPOU
PROGRAM prgBattery
VAR PERSISTENT
	bEnableBattery				: BOOL;							//{#lynus.ag#()}
	byPrioBattery				: BYTE;							//{#lynus.ag#()}
	lrMaxCapacityBattery		: LREAL;						//{#lynus.ag#()}
	lrCounterBattProd			: LREAL;						//{#lynus.ag#()}
	lrCounterBattCons			: LREAL;						//{#lynus.ag#()}
	b_Enable_TimeControl		: BOOL;							//{#lynus.ag#()}
	rSetPointSwitchOff			: LREAL;						//{#lynus.ag#()}
	by_Min_BatterySOC			: BYTE;							//{#lynus.ag#()}
	by_Max_BatterySOC			: BYTE;							//{#lynus.ag#()}
END_VAR
VAR
	fbBattery					: FB_Xelectrix_Powerbox_v2_2;
	fbBattCounter				: FB_EnergyCounter;
	bIsEnabledBattery			: BOOL;							//{#lynus.ag#()}
	bResetBattery				: BOOL;							//{#lynus.ag#()}
	bSResetBattery				: BOOL;							//{#lynus.ag#()}
	byErrorWarningBattery		: BYTE;							//{#lynus.ag#()}
	dwSOCBattery				: DWORD;						//{#lynus.ag#()}
	rTargetPowerBattery			: REAL;							//{#lynus.ag#()}
	lrPowerBattery				: LREAL;						//{#lynus.ag#()}
	lrActualCapacityBattery		: LREAL;						//{#lynus.ag#()}
	
	int_GridState: INT;											//{#lynus.ag#()}
	int_BatteryState: INT;										//{#lynus.ag#()}
	int_OperatingState: INT;									//{#lynus.ag#()}
	int_ErrorState: INT;										//{#lynus.ag#()}

	FB_Interval: FB_IntervalBit;
	m_IslandOperationStart: BOOL;								//{#lynus.ag#()}
	m_IslandOperationOngoing: BOOL;								//{#lynus.ag#()}
	m_IslandOperationStop: BOOL;								//{#lynus.ag#()}
	t_Interval :TIME:=T#30M;
	t_HightTime :TIME:=T#1S;

	m_BatteryErrorActive: BOOL;									//{#lynus.ag#()}
	m_BatteryModbusCommError: BOOL;								//{#lynus.ag#()}
	m_BatteryTargetSPError: BOOL;								//{#lynus.ag#()}
	Ton_Delay_BatteryError: Ton;
	Ton_Delay_BatteryModbusError: Ton;
	Ton_Delay_BatterySPError: Ton;	

	mtest: BOOL;
	x: REAL;
	b_TimeControl_Start			:BOOL;								//{#lynus.ag#()}
	b_TimeControl_Stop			:BOOL;								//{#lynus.ag#()}

	r_Trig_Stop_Battery: R_trig;
	r_Trig_Start_Battery: R_trig;
	rs_Stop_Battery: Rs;
	ton_StopBattery_MainsDelay	:ton;
	byBatteryIslandOperation	: BOOL;								//{#lynus.ag#()}
	byBatteryBypassOperation	: BOOL;								//{#lynus.ag#()}
	by_S_Min_BatterySOC			: BYTE;							//{#lynus.ag#()}
	by_S_Max_BatterySOC			: BYTE;							//{#lynus.ag#()}
END_VAR

IF mtest THEN
	Lynus_Standards.GVL_Energy.stDataOfBatteryInverters[1,1].rTargetPowerEMS:=x;
END_IF

fbBattery(
	bEnable:= bEnableBattery, 
	bActivateControl:= TRUE, 
	byUnitID:= 1, 
	byPriority:= byPrioBattery, 
	diNrOfEMS_IN:= prgEMS.fbEMS.diNrOfEMS_OUT, 
	lrMaxCapacityBattery:= lrMaxCapacityBattery, 
	sIPAdress:= '172.16.127.130', 
	bReset:= bResetBattery, 
	by_minDischargeSOC := by_Min_BatterySOC,
	by_maxChargeSOC := by_Max_BatterySOC,
	m_ManualSetpointEnable:= , 
	i_SetpointPower_Manual_kW:= , 
	m_ManualChargeDischargeMax:= , 
	r_MaxChargePower_W:= , 
	r_MaxDischargePower_W:= , 
	m_go_to_online:= r_Trig_Start_Battery.Q, 
	m_go_to_bypass:= r_Trig_Stop_Battery.Q, 
	stDataXelectrix=> , 
	stDataBatt=> , 
	stDataBattInverter=> , 
	stDataEMPower_Grid=> , 
	stDataEMCounter_Grid=> , 
	diNrOfBatt_OUT=> , 
	diNrOfBattInverter_OUT=> , 
	diNrOfEM_OUT_Grid=> , 
	lrMaxCapacityBattery_OUT=> , 
	iSetpointPower_Info=>  ,
	dw_BatterySOC_notZero=>	,
	by_SminDischargeSOC	=>  by_S_Min_BatterySOC,	
	by_SmaxChargeSOC=> by_S_Max_BatterySOC
);


//Out
bIsEnabledBattery := fbBattery.stDataBatt.bEnabled;
bSResetBattery := fbBattery.stDataBattInverter.bStateReset;
dwSOCBattery := fbBattery.dw_BatterySOC_notZero;						// was original fbBattery.stDataBatt.dwSOC; 	this now shows the last received SOC <> 0
rTargetPowerBattery := fbBattery.stDataBattInverter.rTargetPower;
lrPowerBattery := fbBattery.stDataBatt.lrPower;
lrActualCapacityBattery := fbBattery.stDataBatt.lrCapacity;
byErrorWarningBattery := fbBattery.stDataBatt.byErrorWarning;


// EnergyCounter
fbBattCounter(
	byActiveTariff:= 1, 
	lrPowerInput:= lrPowerBattery, 
	lrTotalCounterEnergy_Consumption=> , 
	lrTotalCounterEnergy_Production=> , 
	lrCounterEnergyT1_Consumption=> , 
	lrCounterEnergyT2_Consumption=> , 
	lrCounterEnergyT1_Production=> , 
	lrCounterEnergyT2_Production=> );
	
IF fbBattCounter.lrTotalCounterEnergy_Production > lrCounterBattProd THEN  	
	lrCounterBattProd := fbBattCounter.lrTotalCounterEnergy_Production;
END_IF

IF fbBattCounter.lrTotalCounterEnergy_Consumption > lrCounterBattCons THEN  	
	lrCounterBattCons := fbBattCounter.lrTotalCounterEnergy_Consumption;
END_IF

// send e states to cloud
int_GridState 		:= fbBattery.stDataXelectrix.eGridState;
int_BatteryState	:= fbBattery.stDataXelectrix.eBatteryState;
int_OperatingState	:= fbBattery.stDataXelectrix.eOperatingState;
int_ErrorState		:= fbBattery.stDataXelectrix.eErrorState;

// create bits when battery is in island operation

FB_Interval(
	m_Input			:=  prgBattery.fbBattery.stDataXelectrix.eGridState = 2,	//   2 = Island Mode 
	t_Interval 		:= t_Interval , 
	t_HighTime		:= t_HightTime, 
	m_RisingEdge	=> m_IslandOperationStart, 
	m_Interval		=> m_IslandOperationOngoing, 
	m_FallingEdge	=> m_IslandOperationStop);
	
// monitoring Battery status

Ton_Delay_BatteryError (In := fbBattery.stDataXelectrix.eErrorState =2,
						PT :=T#5S,
						Q => m_BatteryErrorActive);

Ton_Delay_BatteryModbusError (	In := fbBattery.stDataXelectrix.eErrorState = 1,
								PT :=T#10M,
								Q => m_BatteryModbusCommError);						

Ton_Delay_BatterySPError (	In := ABS(fbBattery.iSetpointPower/10-lrPowerBattery) > 20 AND fbBattery.stDataXelectrix.eGridState<>2 AND fbBattery.stDataBatt.dwSOC<90,	// not alarming during island operation
							PT :=T#1M,
							Q => m_BatteryTargetSPError);		

							(*

// control battery offline
	
r_Trig_Start_Battery(CLK := b_TimeControl_Start AND b_Enable_TimeControl);	

rs_Stop_Battery	(	SET:= b_TimeControl_Stop AND b_Enable_TimeControl, 
					RESET1:= r_Trig_Stop_Battery.Q OR NOT b_Enable_TimeControl, 
					Q1=> );
rSetPointSwitchOff := LIMIT(5,rSetPointSwitchOff,100);
ton_StopBattery_MainsDelay(	IN:= prgHouse.lrPowerHouse < rSetPointSwitchOff, 
							PT:= T#15M, 
							Q=> , 
							ET=> );
r_Trig_Stop_Battery(CLK := rs_Stop_Battery.Q1 AND ton_StopBattery_MainsDelay.Q AND b_Enable_TimeControl);


byBatteryIslandOperation := fbBattery.stDataXelectrix.eGridState=2;
byBatteryBypassOperation := NOT (fbBattery.stDataXelectrix.eBatteryState=4 OR fbBattery.stDataXelectrix.eBatteryState=5); 

*)

END_PROGRAM

// ---- POUs/prgRWEffIO.TcPOU
PROGRAM prgRWEffIO
VAR
	fbRW1		: FB_ReadWrite_V2;
(*	fbRW2		: FB_ReadWrite_V2;
	fbRW3		: FB_ReadWrite_V2;  *)
END_VAR

fbRW1(	eUploadType := eSelectDataUploadType.e_Change_Intervall5min,
		bBusy=> , 
		bError=> , 
		udiErrorCodeOut=> , 
		eErrorReadWrite_Out=> );
(*		
fbRW2(	eUploadType:= eSelectDataUploadType.e_Change_noIntervall, 
		bBusy=> , 
		bError=> , 
		udiErrorCodeOut=> , 
		eErrorReadWrite_Out=> );
		
fbRW3(	eUploadType:=eSelectDataUploadType.e_Change_noIntervall, 
		bBusy=> , 
		bError=> , 
		udiErrorCodeOut=> , 
		eErrorReadWrite_Out=> );
		
		*)

END_PROGRAM

// ---- POUs/prgVarEffIO.TcPOU
PROGRAM prgVarEffIO
VAR
	fbVar		: FB_VarInfo_V3;
END_VAR

fbVar(
	bReadInfo:= , 
	eTMCFile:= eSelectTMCFile.eDontUseTMCFile, 
	eSavePositionTMCFile:= eSavePositionOnPLC.ePostionHardDisk, 
	udiCounterFoundVariables=> , 
	bError=> , 
	bBusy=> , 
	byProgress=> , 
	udiErrorCodeOut=> , 
	eErrorVarInfo_Out=> , 
	sVarWithError=> );

fbVar(
	bReadInfo:= , 
	eTMCFile:= eSelectTMCFile.eDontUseTMCFile, 
	eSavePositionTMCFile:= eSavePositionOnPLC.ePostionHardDisk, 
	udiCounterFoundVariables=> , 
	bError=> , 
	bBusy=> , 
	byProgress=> , 
	udiErrorCodeOut=> , 
	eErrorVarInfo_Out=> , 
	sVarWithError=> );

END_PROGRAM

// ---- POUs/prgComEffIO.TcPOU
PROGRAM prgComEffIO
VAR
	fbCom		: FB_MqttCommunicator_V3;
END_VAR

fbCom(
	bConnect				:= TRUE,
	strAuthKey				:=  'BMS99299754422' , 
	sUserName				:= '3e50e6d5-eb07-43c8-8301-26b96effcdd6', 
	sUserPassword			:= '00b28941-9e96-4cb2-9f19-540a3e4b2bd2', 
	eSavePositionCertificate:= eSavePositionOnPLC.ePostionHardDisk, 
	time_HeartBeat_sec := T#15S,
	bConnected=> , 
	bError=> , 
	hrErrorCode=> , 
	eConnectionState=> , 
	eErrorMessage_Out=> );

END_PROGRAM

// ---- FB/FB_TCPModbusRequest_PV.TcPOU
FUNCTION_BLOCK FB_TCPModbusRequest_PV
VAR_INPUT
	b_Enable: BOOL;
	by_slave_ID	:BYTE;
	str_IPAdress: STRING(15);
	
		
END_VAR
VAR_OUTPUT

	lreal_RealPower_kW:LREAL;
	lreal_Voltage_L1L2_V: LREAL;
	lreal_Voltage_L2L3_V: LREAL;
	lreal_Voltage_L3L1_V: LREAL;
	lreal_Voltage_L1_V: LREAL;
	lreal_Voltage_L2_V: LREAL;
	lreal_Voltage_L3_V: LREAL;
	lreal_Current_L1_A: LREAL;
	lreal_Current_L2_A: LREAL;
	lreal_Current_L3_A: LREAL;
	lreal_PeakPowerDay_kW: LREAL;
	lreal_Power2_kW: LREAL;
	lreal_ReactivePower_kVAr: LREAL;
	lreal_PowerFactor: LREAL;
	lreal_Frequency_Hz: LREAL;
	lreal_Efficiency: LREAL;
	lreal_InternalTemperature_C: LREAL;
	lreal_IsolationResistance_MOhm: LREAL;
END_VAR
VAR
	i_State:INT;
	FB_SocketConnect : FB_SocketConnect;
	hSocket : T_HSOCKET;
	FB_SocketSend : FB_SocketSend;
	FB_SocketReceive : FB_SocketReceive;
	byteSendString : ARRAY[1..12] OF BYTE;
	FB_CloseSockets: FB_SocketCloseAll;
	
	ton_TimeOut: Ton;
	ton_WaitforReconnect: Ton;
	ton_ConnectionEstablised: Ton;
	time_ReconnectTime:TIME:=T#30M;
	b_configured: BOOL;
	byteReceiveString : ARRAY[1..200] OF BYTE;
	FB_BYTE_TO_WORD_1 : FB_CV_BYTE_TO_WORD;
	FB_BYTE_TO_WORD_2 : FB_CV_BYTE_TO_WORD;
	FB_WORD_TO_INT : FB_CV_WORD_TO_INT;
	ton_WaitforNetxtRequest: Ton;
	ton_Wait: Ton;
	int_SuccessCounter: INT;
	int_ReconnectCounter: INT;
	int_ErrorCount: INT;
	fbConvertWordToDword		: FB_CV_WORD_TO_DWORD;			//Convert Word to Dword
	fb_ConvertBytesToLreal		:fb_Convert4BytesToLreal;

END_VAR





IF NOT b_Enable THEN			// go to state 0 if not enabled
	i_State := 0;
END_IF


CASE i_State OF
	0:	// wait for enable state
		IF b_Enable THEN
			i_State := 1;
		END_IF
		FB_SocketConnect.bExecute := FALSE;
		FB_SocketSend.bExecute := FALSE;
		FB_SocketSend.bExecute := FALSE;
		ton_TimeOut.IN :=FALSE;	
		ton_ConnectionEstablised.IN := FALSE;
	

	1: // check if configured
		IF b_configured = FALSE THEN
			// request FC3, Register 32064, 25 Words --> Real PV Power ff
			byteSendString[1] := 0;
			byteSendString[2] := 1;
			byteSendString[3] := 0;
			byteSendString[4] := 0;
			byteSendString[5] := 0;
			byteSendString[6] := 6;
			byteSendString[7] := LIMIT(1,by_slave_ID,255);			// slave id
			byteSendString[8] := 3;
			byteSendString[9] := 125;
			byteSendString[10] := 64;
			byteSendString[11] := 0;
			byteSendString[12] := 25;
		
			b_configured := TRUE;
		END_IF
		i_State := i_State+1;
		
	2: // open socket
		FB_SocketConnect.bExecute := TRUE;
		ton_TimeOut.IN :=TRUE;
		i_State := i_State+1;
		
	3: // wait for connection established	
		IF NOT FB_SocketConnect.bBusy AND NOT FB_SocketConnect.bError THEN
			ton_TimeOut.IN :=FALSE;
			ton_ConnectionEstablised.IN := TRUE;
			i_State := i_State+1;
		ELSIF FB_SocketConnect.bError OR ton_TimeOut.Q THEN
			ton_TimeOut.IN :=FALSE;
			i_State := 100;
		END_IF
	
	4: //connection established, request data
		ton_Wait.IN := TRUE;
		IF ton_Wait.Q THEN
			FB_SocketSend.bExecute := TRUE;
			ton_TimeOut.IN :=TRUE;
			ton_Wait.IN := FALSE;
			i_State := i_State+1;
		END_IF
	
	5: // wait for request sent
		IF NOT FB_SocketSend.bBusy AND NOT FB_SocketSend.bError THEN
			ton_TimeOut.IN :=FALSE;
			FB_SocketSend.bExecute := FALSE;
			i_State := i_State+1;  
		ELSIF FB_SocketSend.bError OR ton_TimeOut.Q THEN
			FB_SocketSend.bExecute := FALSE;
			ton_TimeOut.IN :=FALSE;
			i_State := 100;
		END_IF
		
	6: // wait for data
		ton_Wait.IN := TRUE;
		IF ton_Wait.Q THEN
			FB_SocketReceive.bExecute := TRUE;
			ton_Wait.IN := FALSE;
			i_State := i_State+1; 
		END_IF		 
	
	7:	
		ton_Wait.IN := TRUE;
		IF ton_Wait.Q THEN
			ton_TimeOut.IN :=TRUE;
			i_State := i_State+1; 
		END_IF	
	
	8: // convert received data
		IF NOT FB_SocketReceive.bBusy AND NOT FB_SocketReceive.bError THEN
			int_SuccessCounter := int_SuccessCounter+1;
			ton_TimeOut.IN :=FALSE;
			FB_SocketReceive.bExecute := FALSE;
	
			FB_BYTE_TO_WORD_1(byInputValue_1 := byteReceiveString[14],byInputValue_2 := byteReceiveString[15], Ebyteorderforconvert := Ebyteorder.EBIGENDIAN, woutputvalue => );
			lreal_Voltage_L1L2_V := WORD_TO_LREAL(FB_BYTE_TO_WORD_1.woutputvalue)/10;
			FB_BYTE_TO_WORD_1(byInputValue_1 := byteReceiveString[16],byInputValue_2 := byteReceiveString[17], Ebyteorderforconvert := Ebyteorder.EBIGENDIAN, woutputvalue => );
			lreal_Voltage_L2L3_V := WORD_TO_LREAL(FB_BYTE_TO_WORD_1.woutputvalue)/10;
			FB_BYTE_TO_WORD_1(byInputValue_1 := byteReceiveString[18],byInputValue_2 := byteReceiveString[19], Ebyteorderforconvert := Ebyteorder.EBIGENDIAN, woutputvalue => );
			lreal_Voltage_L3L1_V := WORD_TO_LREAL(FB_BYTE_TO_WORD_1.woutputvalue)/10;
			FB_BYTE_TO_WORD_1(byInputValue_1 := byteReceiveString[20],byInputValue_2 := byteReceiveString[21], Ebyteorderforconvert := Ebyteorder.EBIGENDIAN, woutputvalue => );
			lreal_Voltage_L1_V := WORD_TO_LREAL(FB_BYTE_TO_WORD_1.woutputvalue)/10;
			FB_BYTE_TO_WORD_1(byInputValue_1 := byteReceiveString[22],byInputValue_2 := byteReceiveString[23], Ebyteorderforconvert := Ebyteorder.EBIGENDIAN, woutputvalue => );
			lreal_Voltage_L2_V := WORD_TO_LREAL(FB_BYTE_TO_WORD_1.woutputvalue)/10;
			FB_BYTE_TO_WORD_1(byInputValue_1 := byteReceiveString[24],byInputValue_2 := byteReceiveString[25], Ebyteorderforconvert := Ebyteorder.EBIGENDIAN, woutputvalue => );
			lreal_Voltage_L3_V := WORD_TO_LREAL(FB_BYTE_TO_WORD_1.woutputvalue)/10;


			fb_ConvertBytesToLreal(	by_InputValue_1:= byteReceiveString[10], 
									by_InputValue_2:= byteReceiveString[11], 
									by_InputValue_3:= byteReceiveString[12], 
									by_InputValue_4:= byteReceiveString[13], 
									int_Divider:= 1000, 
									lreal_Output=> );
					
			IF fb_ConvertBytesToLreal.lreal_Output < 100 AND fb_ConvertBytesToLreal.lreal_Output > -1 THEN
				lreal_RealPower_kW := fb_ConvertBytesToLreal.lreal_Output;
			END_IF
			
			fb_ConvertBytesToLreal(	by_InputValue_1:= byteReceiveString[26], 
									by_InputValue_2:= byteReceiveString[27], 
									by_InputValue_3:= byteReceiveString[28], 
									by_InputValue_4:= byteReceiveString[29], 
									int_Divider:= 1000, 
									lreal_Output=> lreal_Current_L1_A);
									
			fb_ConvertBytesToLreal(	by_InputValue_1:= byteReceiveString[30], 
									by_InputValue_2:= byteReceiveString[31], 
									by_InputValue_3:= byteReceiveString[32], 
									by_InputValue_4:= byteReceiveString[33], 
									int_Divider:= 1000, 
									lreal_Output=> lreal_Current_L2_A);

			fb_ConvertBytesToLreal(	by_InputValue_1:= byteReceiveString[34], 
									by_InputValue_2:= byteReceiveString[35], 
									by_InputValue_3:= byteReceiveString[36], 
									by_InputValue_4:= byteReceiveString[37], 
									int_Divider:= 1000, 
									lreal_Output=> lreal_Current_L3_A);
									
			fb_ConvertBytesToLreal(	by_InputValue_1:= byteReceiveString[38], 
									by_InputValue_2:= byteReceiveString[39], 
									by_InputValue_3:= byteReceiveString[40], 
									by_InputValue_4:= byteReceiveString[41], 
									int_Divider:= 1000, 
									lreal_Output=> lreal_PeakPowerDay_kW );

			fb_ConvertBytesToLreal(	by_InputValue_1:= byteReceiveString[42], 
									by_InputValue_2:= byteReceiveString[43], 
									by_InputValue_3:= byteReceiveString[44], 
									by_InputValue_4:= byteReceiveString[45], 
									int_Divider:= 1000, 
									lreal_Output=> lreal_Power2_kW);
			
			fb_ConvertBytesToLreal(	by_InputValue_1:= byteReceiveString[46], 
									by_InputValue_2:= byteReceiveString[47], 
									by_InputValue_3:= byteReceiveString[48], 
									by_InputValue_4:= byteReceiveString[49], 
									int_Divider:= 1000, 
									lreal_Output=>lreal_ReactivePower_kVAr );

			FB_BYTE_TO_WORD_1(byInputValue_1 := byteReceiveString[50],byInputValue_2 := byteReceiveString[51], Ebyteorderforconvert := Ebyteorder.EBIGENDIAN, woutputvalue => );
			lreal_PowerFactor := WORD_TO_LREAL(FB_BYTE_TO_WORD_1.woutputvalue)/1000;
			FB_BYTE_TO_WORD_1(byInputValue_1 := byteReceiveString[52],byInputValue_2 := byteReceiveString[53], Ebyteorderforconvert := Ebyteorder.EBIGENDIAN, woutputvalue => );
			lreal_Frequency_Hz := WORD_TO_LREAL(FB_BYTE_TO_WORD_1.woutputvalue)/100;
			FB_BYTE_TO_WORD_1(byInputValue_1 := byteReceiveString[54],byInputValue_2 := byteReceiveString[55], Ebyteorderforconvert := Ebyteorder.EBIGENDIAN, woutputvalue => );
			lreal_Efficiency := WORD_TO_LREAL(FB_BYTE_TO_WORD_1.woutputvalue)/100;
			FB_BYTE_TO_WORD_1(byInputValue_1 := byteReceiveString[56],byInputValue_2 := byteReceiveString[57], Ebyteorderforconvert := Ebyteorder.EBIGENDIAN, woutputvalue => );
			lreal_InternalTemperature_C := WORD_TO_LREAL(FB_BYTE_TO_WORD_1.woutputvalue)/10;
			FB_BYTE_TO_WORD_1(byInputValue_1 := byteReceiveString[58],byInputValue_2 := byteReceiveString[59], Ebyteorderforconvert := Ebyteorder.EBIGENDIAN, woutputvalue => );
			lreal_IsolationResistance_MOhm := WORD_TO_LREAL(FB_BYTE_TO_WORD_1.woutputvalue)/1000;

		
			//FB_WORD_TO_INT(wInputValue := FB_BYTE_TO_WORD.woutputvalue, iOutputValue => );
			//lreal_RealPower_kW := (INT_TO_LREAL(FB_WORD_TO_INT.iOutputValue))/1000;

			i_State := i_State+1;
		ELSIF FB_SocketSend.bError OR ton_TimeOut.Q THEN
 			FB_SocketReceive.bExecute := FALSE;
			ton_TimeOut.IN :=FALSE;
			i_State := 100;
		END_IF
	
	9: // for for next request
		ton_WaitforNetxtRequest.IN := TRUE;
		IF NOT b_Enable THEN
			ton_WaitforNetxtRequest.IN := FALSE;
			i_State := 10;
		END_IF
		IF ton_WaitforNetxtRequest.Q THEN
			ton_WaitforNetxtRequest.IN := FALSE;
			i_State := 4;
		END_IF
		IF 	ton_ConnectionEstablised.Q THEN 
			ton_WaitforNetxtRequest.IN := FALSE;
			i_State := 10;
		END_IF

	10: // close sockets
		FB_CloseSockets.bExecute := TRUE;
		ton_TimeOut.IN :=TRUE;
		i_State := i_State+1;
		
	11: // wait for sockets closed
		
		IF NOT FB_CloseSockets.bBusy THEN
			int_ReconnectCounter := int_ReconnectCounter+1;
			FB_CloseSockets.bExecute := FALSE;
			i_State := 0;
		ELSIF FB_CloseSockets.bError THEN
			int_ReconnectCounter := int_ReconnectCounter+1;
			FB_CloseSockets.bExecute := FALSE;
			i_State := 0;
		END_IF

	100: // wait state for reconect
		
		FB_SocketConnect.bExecute := FALSE;
		FB_SocketSend.bExecute := FALSE;
		FB_SocketReceive.bExecute := FALSE;
		ton_ConnectionEstablised.IN := FALSE;
		ton_TimeOut.IN :=FALSE;
		ton_WaitforReconnect.IN := TRUE;
		IF ton_WaitforReconnect.Q THEN
			int_ErrorCount := int_ErrorCount+1;
			ton_WaitforReconnect.IN := FALSE;
			i_State := 10;
		END_IF
	
END_CASE



FB_SocketConnect(
	sSrvNetId := '',
	sRemoteHost := str_IPAdress,
	nRemotePort := 502,
	bExecute := ,
	tTimeout := T#1S,
	bBusy =>,
	bError =>,
	nErrId =>,
	hSocket => hSocket);
	
FB_SocketSend(
	sSrvNetId:= '', 
	hSocket:= hSocket, 
	cbLen:= 12,
	pSrc:= ADR( byteSendString ), 
	bExecute:= , 
	tTimeout:= T#3S, 
	bBusy=> , 
	bError=> , 
	nErrId=> );
	
FB_SocketReceive(
	sSrvNetId:= '', 
	hSocket:= hSocket, 
	cbLen:= 200, 
	pDest:= ADR( byteReceiveString ), 
	bExecute:= , 
	tTimeout:= T#3S, 
	bBusy=> , 
	bError=> , 
	nErrId=> , 
	nRecBytes=> );

FB_CloseSockets(
	sSrvNetId:= '', 
	bExecute:= , 
	tTimeout:= T#2S, 
	bBusy=> , 
	bError=> , 
	nErrId=> );
	
ton_TimeOut(PT := T#5S);
ton_WaitforReconnect(PT := T#10S);
ton_ConnectionEstablised(pt := time_ReconnectTime);
ton_WaitforNetxtRequest(PT:= T#10S);
ton_Wait(PT:=T#2S);

END_FUNCTION_BLOCK
